LIN {X 0,Y 303.46,Z 323.911,A -85,B 0,C 180,E1 -16452.825,E2 -16452.825} C_VEL
LIN {X 0,Y 302.118,Z 332.035,A -85,B 0,C 180,E1 -16454.483,E2 -16454.483} C_VEL
LIN {X 0,Y 300.639,Z 339.994,A -85,B 0,C 180,E1 -16456.481,E2 -16456.481} C_VEL
LIN {X 0,Y 299.435,Z 346.378,A -85,B 0,C 180,E1 -16458.492,E2 -16458.492} C_VEL
LIN {X 0,Y 298.527,Z 351.434,A -85,B 0,C 180,E1 -16460.514,E2 -16460.514} C_VEL
LIN {X 0,Y 298.006,Z 354.562,A -85,B 0,C 180,E1 -16462.099,E2 -16462.099} C_VEL
LIN {X 0,Y 297.368,Z 358.253,A -85,B 0,C 180,E1 -16464.575,E2 -16464.575} C_VEL
LIN {X 0,Y 297.174,Z 359.637,A -85,B 0,C 180,E1 -16465.931,E2 -16465.931} C_VEL
LIN {X 0,Y 296.944,Z 361.227,A -85,B 0,C 180,E1 -16468.644,E2 -16468.644} C_VEL
LIN {X 0,Y 296.928,Z 361.456,A -85,B 0,C 180,E1 -16470,E2 -16470} C_VEL
LIN {X 0,Y 296.943,Z 361.266,A -85,B 0,C 180,E1 -16471.356,E2 -16471.356} C_VEL
LIN {X 0,Y 297.157,Z 359.726,A -85,B 0,C 180,E1 -16474.069,E2 -16474.069} C_VEL
LIN {X 0,Y 297.357,Z 358.38,A -85,B 0,C 180,E1 -16475.425,E2 -16475.425} C_VEL
LIN {X 0,Y 297.953,Z 354.9,A -85,B 0,C 180,E1 -16477.826,E2 -16477.826} C_VEL
LIN {X 0,Y 298.756,Z 350.121,A -85,B 0,C 180,E1 -16480.162,E2 -16480.162} C_VEL
LIN {X 0,Y 299.99,Z 343.715,A -85,B 0,C 180,E1 -16482.515,E2 -16482.515} C_VEL
LIN {X 0,Y 301.265,Z 336.671,A -85,B 0,C 180,E1 -16484.524,E2 -16484.524} C_VEL
LIN {X 0,Y 302.83,Z 327.889,A -85,B 0,C 180,E1 -16486.517,E2 -16486.517} C_VEL
LIN {X 0,Y 304.365,Z 318.867,A -85,B 0,C 180,E1 -16488.163,E2 -16488.163} C_VEL
LIN {X 0,Y 305.711,Z 308.49,A -85,B 0,C 180,E1 -16489.7,E2 -16489.7} C_VEL
LIN {X 0,Y 307.133,Z 297.75,A -85,B 0,C 180,E1 -16490.949,E2 -16490.949} C_VEL
LIN {X 0,Y 307.473,Z 294.559,A -85,B 0,C 180,E1 -16491.276,E2 -16491.276} C_VEL
LIN {X 0,Y 305.517,Z 284.175,A -85,B 0,C 180,E1 -16492.412,E2 -16492.412} C_VEL
LIN {X 0,Y 302.269,Z 271.951,A -85,B 0,C 180,E1 -16493.56,E2 -16493.56} C_VEL
LIN {X 0,Y 297.755,Z 258.35,A -85,B 0,C 180,E1 -16494.625,E2 -16494.625} C_VEL
LIN {X 0,Y 297.811,Z 255.408,A -85,B 0,C 180,E1 -16498.163,E2 -16498.163} C_VEL
LIN {X 0,Y 297.983,Z 252.472,A -85,B 0,C 180,E1 -16501.889,E2 -16501.889} C_VEL
LIN {X 0,Y 297.989,Z 251.752,A -85,B 0,C 180,E1 -16502.851,E2 -16502.851} C_VEL
LIN {X 0,Y 298.161,Z 251.347,A -85,B 0,C 180,E1 -16504.452,E2 -16504.452} C_VEL
LIN {X 0,Y 298.374,Z 251.321,A -85,B 0,C 180,E1 -16507.764,E2 -16507.764} C_VEL
LIN {X 0,Y 298.386,Z 251.316,A -85,B 0,C 180,E1 -16511.261,E2 -16511.261} C_VEL
LIN {X 0,Y 298.355,Z 251.319,A -85,B 0,C 180,E1 -16515.035,E2 -16515.035} C_VEL
LIN {X 0,Y 298.386,Z 251.315,A -85,B 0,C 180,E1 -16518.738,E2 -16518.738} C_VEL
LIN {X 0,Y 298.426,Z 251.311,A -85,B 0,C 180,E1 -16522.243,E2 -16522.243} C_VEL
LIN {X 0,Y 298.41,Z 251.315,A -85,B 0,C 180,E1 -16525.581,E2 -16525.581} C_VEL
LIN {X 0,Y 298.379,Z 251.314,A -85,B 0,C 180,E1 -16528.789,E2 -16528.789} C_VEL
LIN {X 0,Y 298.415,Z 251.312,A -85,B 0,C 180,E1 -16531.899,E2 -16531.899} C_VEL
LIN {X 0,Y 298.441,Z 251.308,A -85,B 0,C 180,E1 -16534.92,E2 -16534.92} C_VEL
LIN {X 0,Y 298.416,Z 251.31,A -85,B 0,C 180,E1 -16537.863,E2 -16537.863} C_VEL
LIN {X 0,Y 298.505,Z 251.301,A -85,B 0,C 180,E1 -16540.754,E2 -16540.754} C_VEL
LIN {X 0,Y 298.587,Z 251.292,A -85,B 0,C 180,E1 -16544.994,E2 -16544.994} C_VEL
LIN {X 0,Y 298.596,Z 251.291,A -85,B 0,C 180,E1 -16549.147,E2 -16549.147} C_VEL
LIN {X 0,Y 298.703,Z 251.276,A -85,B 0,C 180,E1 -16550.695,E2 -16550.695} C_VEL
LIN {X 0,Y 298.097,Z 251.352,A -85,B 0,C 180,E1 -16551.822,E2 -16551.822} C_VEL
LIN {X 0,Y 295.14,Z 251.719,A -85,B 0,C 180,E1 -16553.651,E2 -16553.651} C_VEL
LIN {X 0,Y 292.648,Z 252.03,A -85,B 0,C 180,E1 -16555.138,E2 -16555.138} C_VEL
LIN {X 0,Y 291.677,Z 252.151,A -85,B 0,C 180,E1 -16556.292,E2 -16556.292} C_VEL
LIN {X 0,Y 291.655,Z 252.151,A -85,B 0,C 180,E1 -16556.683,E2 -16556.683} C_VEL
LIN {X 0,Y 291.874,Z 252.13,A -85,B 0,C 180,E1 -16558.62,E2 -16558.62} C_VEL
LIN {X 0,Y 291.889,Z 252.124,A -85,B 0,C 180,E1 -16561.38,E2 -16561.38} C_VEL
LIN {X 0,Y 291.725,Z 252.145,A -85,B 0,C 180,E1 -16566.918,E2 -16566.918} C_VEL
LIN {X 0,Y 291.569,Z 252.164,A -85,B 0,C 180,E1 -16569.714,E2 -16569.714} C_VEL
LIN {X 0,Y 291.523,Z 252.172,A -85,B 0,C 180,E1 -16573.95,E2 -16573.95} C_VEL
LIN {X 0,Y 291.489,Z 252.174,A -85,B 0,C 180,E1 -16576.818,E2 -16576.818} C_VEL
LIN {X 0,Y 291.452,Z 252.182,A -85,B 0,C 180,E1 -16579.875,E2 -16579.875} C_VEL
LIN {X 0,Y 291.335,Z 252.197,A -85,B 0,C 180,E1 -16584.211,E2 -16584.211} C_VEL
LIN {X 0,Y 291.352,Z 252.196,A -85,B 0,C 180,E1 -16587.279,E2 -16587.279} C_VEL
LIN {X 0,Y 291.32,Z 252.199,A -85,B 0,C 180,E1 -16590.439,E2 -16590.439} C_VEL
LIN {X 0,Y 291.345,Z 252.197,A -85,B 0,C 180,E1 -16593.698,E2 -16593.698} C_VEL
LIN {X 0,Y 291.36,Z 252.193,A -85,B 0,C 180,E1 -16597.25,E2 -16597.25} C_VEL
LIN {X 0,Y 291.401,Z 252.404,A -85,B 0,C 180,E1 -16598.619,E2 -16598.619} C_VEL
LIN {X 0,Y 292.148,Z 256.598,A -85,B 0,C 180,E1 -16602.344,E2 -16602.344} C_VEL
LIN {X 0,Y 293.011,Z 261.073,A -85,B 0,C 180,E1 -16606.019,E2 -16606.019} C_VEL
LIN {X 0,Y 293.916,Z 266.185,A -85,B 0,C 180,E1 -16609.922,E2 -16609.922} C_VEL
LIN {X 0,Y 294.31,Z 269.06,A -85,B 0,C 180,E1 -16612.002,E2 -16612.002} C_VEL
LIN {X 0,Y 294.165,Z 272.478,A -85,B 0,C 180,E1 -16614.322,E2 -16614.322} C_VEL
LIN {X 0,Y 293.112,Z 278.393,A -85,B 0,C 180,E1 -16618.163,E2 -16618.163} C_VEL
LIN {X 0,Y 292.122,Z 284.445,A -85,B 0,C 180,E1 -16622.022,E2 -16622.022} C_VEL
LIN {X 0,Y 291.473,Z 288.992,A -85,B 0,C 180,E1 -16624.815,E2 -16624.815} C_VEL
LIN {X 0,Y 294.407,Z 302.447,A -85,B 0,C 180,E1 -16625.676,E2 -16625.676} C_VEL
LIN {X 0,Y 296.405,Z 315.779,A -85,B 0,C 180,E1 -16626.761,E2 -16626.761} C_VEL
LIN {X 0,Y 297.483,Z 327.947,A -85,B 0,C 180,E1 -16627.973,E2 -16627.973} C_VEL
LIN {X 0,Y 297.935,Z 338.759,A -85,B 0,C 180,E1 -16629.278,E2 -16629.278} C_VEL
LIN {X 0,Y 296.165,Z 349.684,A -85,B 0,C 180,E1 -16630.777,E2 -16630.777} C_VEL
LIN {X 0,Y 294.663,Z 358.572,A -85,B 0,C 180,E1 -16632.289,E2 -16632.289} C_VEL
LIN {X 0,Y 293.407,Z 366.829,A -85,B 0,C 180,E1 -16634.011,E2 -16634.011} C_VEL
LIN {X 0,Y 292.021,Z 374.897,A -85,B 0,C 180,E1 -16636.074,E2 -16636.074} C_VEL
LIN {X 0,Y 290.893,Z 381.371,A -85,B 0,C 180,E1 -16638.15,E2 -16638.15} C_VEL
LIN {X 0,Y 290.223,Z 386.529,A -85,B 0,C 180,E1 -16640.241,E2 -16640.241} C_VEL
LIN {X 0,Y 289.817,Z 390.543,A -85,B 0,C 180,E1 -16642.336,E2 -16642.336} C_VEL
LIN {X 0,Y 289.625,Z 393.516,A -85,B 0,C 180,E1 -16644.43,E2 -16644.43} C_VEL
LIN {X 0,Y 289.583,Z 394.933,A -85,B 0,C 180,E1 -16645.825,E2 -16645.825} C_VEL
LIN {X 0,Y 289.557,Z 395.944,A -85,B 0,C 180,E1 -16647.218,E2 -16647.218} C_VEL
LIN {X 0,Y 289.581,Z 396.564,A -85,B 0,C 180,E1 -16648.61,E2 -16648.61} C_VEL
LIN {X 0,Y 289.692,Z 396.788,A -85,B 0,C 180,E1 -16650,E2 -16650} C_VEL
LIN {X 0,Y 289.581,Z 396.559,A -85,B 0,C 180,E1 -16651.391,E2 -16651.391} C_VEL
LIN {X 0,Y 289.557,Z 395.938,A -85,B 0,C 180,E1 -16652.783,E2 -16652.783} C_VEL
LIN {X 0,Y 289.582,Z 394.924,A -85,B 0,C 180,E1 -16654.176,E2 -16654.176} C_VEL
LIN {X 0,Y 289.632,Z 393.206,A -85,B 0,C 180,E1 -16655.802,E2 -16655.802} C_VEL
LIN {X 0,Y 289.906,Z 389.275,A -85,B 0,C 180,E1 -16658.364,E2 -16658.364} C_VEL
LIN {X 0,Y 290.45,Z 384.885,A -85,B 0,C 180,E1 -16660.456,E2 -16660.456} C_VEL
LIN {X 0,Y 291.205,Z 379.299,A -85,B 0,C 180,E1 -16662.545,E2 -16662.545} C_VEL
LIN {X 0,Y 292.467,Z 372.352,A -85,B 0,C 180,E1 -16664.615,E2 -16664.615} C_VEL
LIN {X 0,Y 293.943,Z 363.661,A -85,B 0,C 180,E1 -16666.674,E2 -16666.674} C_VEL
LIN {X 0,Y 295.26,Z 354.749,A -85,B 0,C 180,E1 -16668.385,E2 -16668.385} C_VEL
LIN {X 0,Y 297.11,Z 343.814,A -85,B 0,C 180,E1 -16670.06,E2 -16670.06} C_VEL
LIN {X 0,Y 297.932,Z 338.625,A -85,B 0,C 180,E1 -16670.723,E2 -16670.723} C_VEL
LIN {X 0,Y 297.425,Z 327.766,A -85,B 0,C 180,E1 -16672.032,E2 -16672.032} C_VEL
LIN {X 0,Y 296.354,Z 315.227,A -85,B 0,C 180,E1 -16673.268,E2 -16673.268} C_VEL
LIN {X 0,Y 294.319,Z 301.984,A -85,B 0,C 180,E1 -16674.338,E2 -16674.338} C_VEL
LIN {X 0,Y 291.474,Z 288.763,A -85,B 0,C 180,E1 -16675.197,E2 -16675.197} C_VEL
LIN {X 0,Y 292.497,Z 282.092,A -85,B 0,C 180,E1 -16679.454,E2 -16679.454} C_VEL
LIN {X 0,Y 293.547,Z 275.913,A -85,B 0,C 180,E1 -16683.413,E2 -16683.413} C_VEL
LIN {X 0,Y 294.363,Z 270.985,A -85,B 0,C 180,E1 -16686.647,E2 -16686.647} C_VEL
LIN {X 0,Y 294.104,Z 267.282,A -85,B 0,C 180,E1 -16689.223,E2 -16689.223} C_VEL
LIN {X 0,Y 293.207,Z 262.122,A -85,B 0,C 180,E1 -16693.056,E2 -16693.056} C_VEL
LIN {X 0,Y 292.472,Z 258.342,A -85,B 0,C 180,E1 -16696.129,E2 -16696.129} C_VEL
LIN {X 0,Y 291.749,Z 254.528,A -85,B 0,C 180,E1 -16699.428,E2 -16699.428} C_VEL
LIN {X 0,Y 291.35,Z 252.192,A -85,B 0,C 180,E1 -16701.588,E2 -16701.588} C_VEL
LIN {X 0,Y 291.37,Z 252.191,A -85,B 0,C 180,E1 -16705.095,E2 -16705.095} C_VEL
LIN {X 0,Y 291.369,Z 252.19,A -85,B 0,C 180,E1 -16707.95,E2 -16707.95} C_VEL
LIN {X 0,Y 291.346,Z 252.192,A -85,B 0,C 180,E1 -16711.154,E2 -16711.154} C_VEL
LIN {X 0,Y 291.35,Z 252.196,A -85,B 0,C 180,E1 -16714.266,E2 -16714.266} C_VEL
LIN {X 0,Y 291.356,Z 252.192,A -85,B 0,C 180,E1 -16717.297,E2 -16717.297} C_VEL
LIN {X 0,Y 291.461,Z 252.182,A -85,B 0,C 180,E1 -16720.27,E2 -16720.27} C_VEL
LIN {X 0,Y 291.559,Z 252.166,A -85,B 0,C 180,E1 -16724.624,E2 -16724.624} C_VEL
LIN {X 0,Y 291.532,Z 252.169,A -85,B 0,C 180,E1 -16728.88,E2 -16728.88} C_VEL
LIN {X 0,Y 291.66,Z 252.157,A -85,B 0,C 180,E1 -16731.687,E2 -16731.687} C_VEL
LIN {X 0,Y 291.627,Z 252.157,A -85,B 0,C 180,E1 -16734.468,E2 -16734.468} C_VEL
LIN {X 0,Y 291.891,Z 252.124,A -85,B 0,C 180,E1 -16738.62,E2 -16738.62} C_VEL
LIN {X 0,Y 291.876,Z 252.129,A -85,B 0,C 180,E1 -16741.38,E2 -16741.38} C_VEL
LIN {X 0,Y 291.719,Z 252.146,A -85,B 0,C 180,E1 -16746.919,E2 -16746.919} C_VEL
LIN {X 0,Y 291.572,Z 252.165,A -85,B 0,C 180,E1 -16749.714,E2 -16749.714} C_VEL
LIN {X 0,Y 291.52,Z 252.17,A -85,B 0,C 180,E1 -16753.951,E2 -16753.951} C_VEL
LIN {X 0,Y 291.437,Z 252.184,A -85,B 0,C 180,E1 -16756.821,E2 -16756.821} C_VEL
LIN {X 0,Y 291.427,Z 252.181,A -85,B 0,C 180,E1 -16759.86,E2 -16759.86} C_VEL
LIN {X 0,Y 291.364,Z 252.19,A -85,B 0,C 180,E1 -16764.209,E2 -16764.209} C_VEL
LIN {X 0,Y 291.357,Z 252.191,A -85,B 0,C 180,E1 -16767.278,E2 -16767.278} C_VEL
LIN {X 0,Y 291.321,Z 252.199,A -85,B 0,C 180,E1 -16770.439,E2 -16770.439} C_VEL
LIN {X 0,Y 291.347,Z 252.192,A -85,B 0,C 180,E1 -16773.698,E2 -16773.698} C_VEL
LIN {X 0,Y 291.384,Z 252.187,A -85,B 0,C 180,E1 -16777.255,E2 -16777.255} C_VEL
LIN {X 0,Y 291.337,Z 252.195,A -85,B 0,C 180,E1 -16780.642,E2 -16780.642} C_VEL
LIN {X 0,Y 291.293,Z 252.2,A -85,B 0,C 180,E1 -16784.402,E2 -16784.402} C_VEL
LIN {X 0,Y 291.329,Z 252.196,A -85,B 0,C 180,E1 -16788.404,E2 -16788.404} C_VEL
LIN {X 0,Y 291.337,Z 252.193,A -85,B 0,C 180,E1 -16791.155,E2 -16791.155} C_VEL
LIN {X 0,Y 291.329,Z 252.193,A -85,B 0,C 180,E1 -16792.907,E2 -16792.907} C_VEL
LIN {X 0,Y 291.005,Z 252.237,A -85,B 0,C 180,E1 -16796.257,E2 -16796.257} C_VEL
LIN {X 0,Y 290.906,Z 254.487,A -85,B 0,C 180,E1 -16799.513,E2 -16799.513} C_VEL
LIN {X 0,Y 290.769,Z 257.655,A -85,B 0,C 180,E1 -16803.42,E2 -16803.42} C_VEL
LIN {X 0,Y 290.733,Z 258.839,A -85,B 0,C 180,E1 -16804.862,E2 -16804.862} C_VEL
LIN {X 0,Y 295.305,Z 272.378,A -85,B 0,C 180,E1 -16805.967,E2 -16805.967} C_VEL
LIN {X 0,Y 298.493,Z 284.073,A -85,B 0,C 180,E1 -16807.102,E2 -16807.102} C_VEL
LIN {X 0,Y 300.734,Z 295.59,A -85,B 0,C 180,E1 -16808.403,E2 -16808.403} C_VEL
LIN {X 0,Y 299.32,Z 306.86,A -85,B 0,C 180,E1 -16809.69,E2 -16809.69} C_VEL
LIN {X 0,Y 297.828,Z 317.602,A -85,B 0,C 180,E1 -16811.245,E2 -16811.245} C_VEL
LIN {X 0,Y 296.371,Z 326.109,A -85,B 0,C 180,E1 -16812.757,E2 -16812.757} C_VEL
LIN {X 0,Y 295.071,Z 333.933,A -85,B 0,C 180,E1 -16814.457,E2 -16814.457} C_VEL
LIN {X 0,Y 293.529,Z 341.587,A -85,B 0,C 180,E1 -16816.5,E2 -16816.5} C_VEL
LIN {X 0,Y 292.128,Z 348.604,A -85,B 0,C 180,E1 -16818.903,E2 -16818.903} C_VEL
LIN {X 0,Y 291.296,Z 353.268,A -85,B 0,C 180,E1 -16820.977,E2 -16820.977} C_VEL
LIN {X 0,Y 290.723,Z 356.832,A -85,B 0,C 180,E1 -16823.057,E2 -16823.057} C_VEL
LIN {X 0,Y 290.329,Z 358.68,A -85,B 0,C 180,E1 -16824.443,E2 -16824.443} C_VEL
LIN {X 0,Y 290.104,Z 360.064,A -85,B 0,C 180,E1 -16825.832,E2 -16825.832} C_VEL
LIN {X 0,Y 289.859,Z 361.654,A -85,B 0,C 180,E1 -16828.61,E2 -16828.61} C_VEL
LIN {X 0,Y 289.841,Z 361.882,A -85,B 0,C 180,E1 -16830,E2 -16830} C_VEL
LIN {X 0,Y 289.858,Z 361.692,A -85,B 0,C 180,E1 -16831.389,E2 -16831.389} C_VEL
LIN {X 0,Y 290.088,Z 360.152,A -85,B 0,C 180,E1 -16834.168,E2 -16834.168} C_VEL
LIN {X 0,Y 290.316,Z 358.805,A -85,B 0,C 180,E1 -16835.557,E2 -16835.557} C_VEL
LIN {X 0,Y 290.903,Z 355.549,A -85,B 0,C 180,E1 -16837.889,E2 -16837.889} C_VEL
LIN {X 0,Y 291.775,Z 350.547,A -85,B 0,C 180,E1 -16840.408,E2 -16840.408} C_VEL
LIN {X 0,Y 293.09,Z 344.139,A -85,B 0,C 180,E1 -16842.815,E2 -16842.815} C_VEL
LIN {X 0,Y 294.421,Z 337.095,A -85,B 0,C 180,E1 -16844.869,E2 -16844.869} C_VEL
LIN {X 0,Y 296.051,Z 328.312,A -85,B 0,C 180,E1 -16846.906,E2 -16846.906} C_VEL
LIN {X 0,Y 297.643,Z 319.29,A -85,B 0,C 180,E1 -16848.588,E2 -16848.588} C_VEL
LIN {X 0,Y 298.991,Z 309.413,A -85,B 0,C 180,E1 -16850.091,E2 -16850.091} C_VEL
LIN {X 0,Y 300.524,Z 298.171,A -85,B 0,C 180,E1 -16851.432,E2 -16851.432} C_VEL
LIN {X 0,Y 300.731,Z 294.989,A -85,B 0,C 180,E1 -16851.777,E2 -16851.777} C_VEL
LIN {X 0,Y 298.469,Z 283.823,A -85,B 0,C 180,E1 -16853.037,E2 -16853.037} C_VEL
LIN {X 0,Y 295.243,Z 272.161,A -85,B 0,C 180,E1 -16854.171,E2 -16854.171} C_VEL
LIN {X 0,Y 291.253,Z 260.862,A -85,B 0,C 180,E1 -16855.118,E2 -16855.118} C_VEL
LIN {X 0,Y 290.703,Z 258.773,A -85,B 0,C 180,E1 -16855.288,E2 -16855.288} C_VEL
LIN {X 0,Y 290.864,Z 255.325,A -85,B 0,C 180,E1 -16859.558,E2 -16859.558} C_VEL
LIN {X 0,Y 290.954,Z 253.239,A -85,B 0,C 180,E1 -16862.282,E2 -16862.282} C_VEL
LIN {X 0,Y 291.004,Z 252.239,A -85,B 0,C 180,E1 -16863.743,E2 -16863.743} C_VEL
LIN {X 0,Y 291.317,Z 252.199,A -85,B 0,C 180,E1 -16867.238,E2 -16867.238} C_VEL
LIN {X 0,Y 291.332,Z 252.196,A -85,B 0,C 180,E1 -16870.643,E2 -16870.643} C_VEL
LIN {X 0,Y 291.292,Z 252.201,A -85,B 0,C 180,E1 -16874.402,E2 -16874.402} C_VEL
LIN {X 0,Y 291.328,Z 252.195,A -85,B 0,C 180,E1 -16878.404,E2 -16878.404} C_VEL
LIN {X 0,Y 291.365,Z 252.19,A -85,B 0,C 180,E1 -16881.16,E2 -16881.16} C_VEL
LIN {X 0,Y 291.363,Z 252.19,A -85,B 0,C 180,E1 -16884.626,E2 -16884.626} C_VEL
LIN {X 0,Y 291.368,Z 252.19,A -85,B 0,C 180,E1 -16887.95,E2 -16887.95} C_VEL
LIN {X 0,Y 291.346,Z 252.194,A -85,B 0,C 180,E1 -16891.154,E2 -16891.154} C_VEL
LIN {X 0,Y 291.36,Z 252.189,A -85,B 0,C 180,E1 -16894.266,E2 -16894.266} C_VEL
LIN {X 0,Y 291.372,Z 252.191,A -85,B 0,C 180,E1 -16897.299,E2 -16897.299} C_VEL
LIN {X 0,Y 291.441,Z 252.18,A -85,B 0,C 180,E1 -16900.269,E2 -16900.269} C_VEL
LIN {X 0,Y 291.499,Z 252.174,A -85,B 0,C 180,E1 -16904.665,E2 -16904.665} C_VEL
LIN {X 0,Y 291.539,Z 252.17,A -85,B 0,C 180,E1 -16908.881,E2 -16908.881} C_VEL
LIN {X 0,Y 291.711,Z 252.146,A -85,B 0,C 180,E1 -16911.688,E2 -16911.688} C_VEL
LIN {X 0,Y 291.627,Z 252.159,A -85,B 0,C 180,E1 -16914.468,E2 -16914.468} C_VEL
LIN {X 0,Y 291.655,Z 252.151,A -85,B 0,C 180,E1 -16916.683,E2 -16916.683} C_VEL
LIN {X 0,Y 291.459,Z 252.178,A -85,B 0,C 180,E1 -16917.454,E2 -16917.454} C_VEL
LIN {X 0,Y 290.212,Z 252.337,A -85,B 0,C 180,E1 -16918.594,E2 -16918.594} C_VEL
LIN {X 0,Y 285.906,Z 252.87,A -85,B 0,C 180,E1 -16921.243,E2 -16921.243} C_VEL
LIN {X 0,Y 284.834,Z 253.006,A -85,B 0,C 180,E1 -16922.426,E2 -16922.426} C_VEL
LIN {X 0,Y 284.744,Z 253.015,A -85,B 0,C 180,E1 -16922.827,E2 -16922.827} C_VEL
LIN {X 0,Y 284.676,Z 253.023,A -85,B 0,C 180,E1 -16927.091,E2 -16927.091} C_VEL
LIN {X 0,Y 284.515,Z 253.044,A -85,B 0,C 180,E1 -16929.957,E2 -16929.957} C_VEL
LIN {X 0,Y 284.483,Z 253.049,A -85,B 0,C 180,E1 -16934.303,E2 -16934.303} C_VEL
LIN {X 0,Y 284.427,Z 253.054,A -85,B 0,C 180,E1 -16937.248,E2 -16937.248} C_VEL
LIN {X 0,Y 284.378,Z 253.063,A -85,B 0,C 180,E1 -16940.242,E2 -16940.242} C_VEL
LIN {X 0,Y 284.29,Z 253.074,A -85,B 0,C 180,E1 -16944.851,E2 -16944.851} C_VEL
LIN {X 0,Y 284.282,Z 253.078,A -85,B 0,C 180,E1 -16948.016,E2 -16948.016} C_VEL
LIN {X 0,Y 284.286,Z 253.078,A -85,B 0,C 180,E1 -16951.276,E2 -16951.276} C_VEL
LIN {X 0,Y 284.337,Z 253.069,A -85,B 0,C 180,E1 -16955.347,E2 -16955.347} C_VEL
LIN {X 0,Y 284.345,Z 253.209,A -85,B 0,C 180,E1 -16957.879,E2 -16957.879} C_VEL
LIN {X 0,Y 285.219,Z 258.045,A -85,B 0,C 180,E1 -16962.335,E2 -16962.335} C_VEL
LIN {X 0,Y 286.174,Z 263.074,A -85,B 0,C 180,E1 -16966.557,E2 -16966.557} C_VEL
LIN {X 0,Y 287.051,Z 268.111,A -85,B 0,C 180,E1 -16970.464,E2 -16970.464} C_VEL
LIN {X 0,Y 287.331,Z 271.836,A -85,B 0,C 180,E1 -16973.158,E2 -16973.158} C_VEL
LIN {X 0,Y 286.498,Z 276.801,A -85,B 0,C 180,E1 -16976.517,E2 -16976.517} C_VEL
LIN {X 0,Y 285.43,Z 282.827,A -85,B 0,C 180,E1 -16980.498,E2 -16980.498} C_VEL
LIN {X 0,Y 284.533,Z 288.393,A -85,B 0,C 180,E1 -16984.138,E2 -16984.138} C_VEL
LIN {X 0,Y 287.621,Z 302.816,A -85,B 0,C 180,E1 -16985.114,E2 -16985.114} C_VEL
LIN {X 0,Y 289.477,Z 314.636,A -85,B 0,C 180,E1 -16986.113,E2 -16986.113} C_VEL
LIN {X 0,Y 290.5,Z 325.712,A -85,B 0,C 180,E1 -16987.227,E2 -16987.227} C_VEL
LIN {X 0,Y 291.01,Z 336.89,A -85,B 0,C 180,E1 -16988.577,E2 -16988.577} C_VEL
LIN {X 0,Y 290.884,Z 340.948,A -85,B 0,C 180,E1 -16989.122,E2 -16989.122} C_VEL
LIN {X 0,Y 289.035,Z 351.408,A -85,B 0,C 180,E1 -16990.653,E2 -16990.653} C_VEL
LIN {X 0,Y 287.482,Z 360.33,A -85,B 0,C 180,E1 -16992.28,E2 -16992.28} C_VEL
LIN {X 0,Y 285.982,Z 369.281,A -85,B 0,C 180,E1 -16994.316,E2 -16994.316} C_VEL
LIN {X 0,Y 284.671,Z 376.764,A -85,B 0,C 180,E1 -16996.436,E2 -16996.436} C_VEL
LIN {X 0,Y 283.646,Z 382.781,A -85,B 0,C 180,E1 -16998.567,E2 -16998.567} C_VEL
LIN {X 0,Y 283.031,Z 387.55,A -85,B 0,C 180,E1 -17000.712,E2 -17000.712} C_VEL
LIN {X 0,Y 282.681,Z 391.202,A -85,B 0,C 180,E1 -17002.859,E2 -17002.859} C_VEL
LIN {X 0,Y 282.562,Z 393.089,A -85,B 0,C 180,E1 -17004.29,E2 -17004.29} C_VEL
LIN {X 0,Y 282.503,Z 394.506,A -85,B 0,C 180,E1 -17005.72,E2 -17005.72} C_VEL
LIN {X 0,Y 282.483,Z 395.518,A -85,B 0,C 180,E1 -17007.148,E2 -17007.148} C_VEL
LIN {X 0,Y 282.495,Z 396.137,A -85,B 0,C 180,E1 -17008.575,E2 -17008.575} C_VEL
LIN {X 0,Y 282.602,Z 396.361,A -85,B 0,C 180,E1 -17010,E2 -17010} C_VEL
LIN {X 0,Y 282.483,Z 395.511,A -85,B 0,C 180,E1 -17012.852,E2 -17012.852} C_VEL
LIN {X 0,Y 282.502,Z 394.496,A -85,B 0,C 180,E1 -17014.28,E2 -17014.28} C_VEL
LIN {X 0,Y 282.559,Z 392.986,A -85,B 0,C 180,E1 -17015.782,E2 -17015.782} C_VEL
LIN {X 0,Y 282.74,Z 390.089,A -85,B 0,C 180,E1 -17017.858,E2 -17017.858} C_VEL
LIN {X 0,Y 283.196,Z 386.065,A -85,B 0,C 180,E1 -17020.004,E2 -17020.004} C_VEL
LIN {X 0,Y 284.079,Z 379.888,A -85,B 0,C 180,E1 -17022.502,E2 -17022.502} C_VEL
LIN {X 0,Y 285.342,Z 373.165,A -85,B 0,C 180,E1 -17024.623,E2 -17024.623} C_VEL
LIN {X 0,Y 286.837,Z 364.828,A -85,B 0,C 180,E1 -17026.732,E2 -17026.732} C_VEL
LIN {X 0,Y 288.178,Z 356.278,A -85,B 0,C 180,E1 -17028.484,E2 -17028.484} C_VEL
LIN {X 0,Y 289.825,Z 346.923,A -85,B 0,C 180,E1 -17030.031,E2 -17030.031} C_VEL
LIN {X 0,Y 291.077,Z 339.515,A -85,B 0,C 180,E1 -17031.049,E2 -17031.049} C_VEL
LIN {X 0,Y 290.66,Z 328.144,A -85,B 0,C 180,E1 -17032.486,E2 -17032.486} C_VEL
LIN {X 0,Y 289.617,Z 315.766,A -85,B 0,C 180,E1 -17033.761,E2 -17033.761} C_VEL
LIN {X 0,Y 287.603,Z 302.612,A -85,B 0,C 180,E1 -17034.878,E2 -17034.878} C_VEL
LIN {X 0,Y 284.779,Z 290.047,A -85,B 0,C 180,E1 -17035.748,E2 -17035.748} C_VEL
LIN {X 0,Y 284.525,Z 288.292,A -85,B 0,C 180,E1 -17035.863,E2 -17035.863} C_VEL
LIN {X 0,Y 285.428,Z 282.785,A -85,B 0,C 180,E1 -17039.502,E2 -17039.502} C_VEL
LIN {X 0,Y 286.498,Z 276.76,A -85,B 0,C 180,E1 -17043.483,E2 -17043.483} C_VEL
LIN {X 0,Y 287.345,Z 271.792,A -85,B 0,C 180,E1 -17046.841,E2 -17046.841} C_VEL
LIN {X 0,Y 287.041,Z 268.049,A -85,B 0,C 180,E1 -17049.539,E2 -17049.539} C_VEL
LIN {X 0,Y 286.145,Z 263.016,A -85,B 0,C 180,E1 -17053.449,E2 -17053.449} C_VEL
LIN {X 0,Y 285.438,Z 259.423,A -85,B 0,C 180,E1 -17056.416,E2 -17056.416} C_VEL
LIN {X 0,Y 284.709,Z 255.313,A -85,B 0,C 180,E1 -17060.073,E2 -17060.073} C_VEL
LIN {X 0,Y 284.326,Z 253.071,A -85,B 0,C 180,E1 -17062.278,E2 -17062.278} C_VEL
LIN {X 0,Y 284.309,Z 253.07,A -85,B 0,C 180,E1 -17065.351,E2 -17065.351} C_VEL
LIN {X 0,Y 284.288,Z 253.075,A -85,B 0,C 180,E1 -17068.725,E2 -17068.725} C_VEL
LIN {X 0,Y 284.284,Z 253.074,A -85,B 0,C 180,E1 -17071.984,E2 -17071.984} C_VEL
LIN {X 0,Y 284.301,Z 253.074,A -85,B 0,C 180,E1 -17076.158,E2 -17076.158} C_VEL
LIN {X 0,Y 284.391,Z 253.062,A -85,B 0,C 180,E1 -17079.898,E2 -17079.898} C_VEL
LIN {X 0,Y 284.496,Z 253.047,A -85,B 0,C 180,E1 -17084.459,E2 -17084.459} C_VEL
LIN {X 0,Y 284.485,Z 253.047,A -85,B 0,C 180,E1 -17088.601,E2 -17088.601} C_VEL
LIN {X 0,Y 284.605,Z 253.034,A -85,B 0,C 180,E1 -17091.48,E2 -17091.48} C_VEL
LIN {X 0,Y 284.597,Z 253.033,A -85,B 0,C 180,E1 -17094.331,E2 -17094.331} C_VEL
LIN {X 0,Y 284.858,Z 253,A -85,B 0,C 180,E1 -17098.586,E2 -17098.586} C_VEL
LIN {X 0,Y 284.843,Z 253.005,A -85,B 0,C 180,E1 -17101.414,E2 -17101.414} C_VEL
LIN {X 0,Y 284.672,Z 253.025,A -85,B 0,C 180,E1 -17107.091,E2 -17107.091} C_VEL
LIN {X 0,Y 284.518,Z 253.042,A -85,B 0,C 180,E1 -17109.957,E2 -17109.957} C_VEL
LIN {X 0,Y 284.467,Z 253.049,A -85,B 0,C 180,E1 -17114.304,E2 -17114.304} C_VEL
LIN {X 0,Y 284.366,Z 253.063,A -85,B 0,C 180,E1 -17118.741,E2 -17118.741} C_VEL
LIN {X 0,Y 284.317,Z 253.067,A -85,B 0,C 180,E1 -17121.764,E2 -17121.764} C_VEL
LIN {X 0,Y 284.309,Z 253.071,A -85,B 0,C 180,E1 -17124.849,E2 -17124.849} C_VEL
LIN {X 0,Y 284.287,Z 253.072,A -85,B 0,C 180,E1 -17128.016,E2 -17128.016} C_VEL
LIN {X 0,Y 284.288,Z 253.071,A -85,B 0,C 180,E1 -17131.275,E2 -17131.275} C_VEL
LIN {X 0,Y 284.344,Z 253.063,A -85,B 0,C 180,E1 -17135.348,E2 -17135.348} C_VEL
LIN {X 0,Y 284.322,Z 253.071,A -85,B 0,C 180,E1 -17138.168,E2 -17138.168} C_VEL
LIN {X 0,Y 284.272,Z 253.075,A -85,B 0,C 180,E1 -17142.124,E2 -17142.124} C_VEL
LIN {X 0,Y 284.259,Z 253.078,A -85,B 0,C 180,E1 -17146.189,E2 -17146.189} C_VEL
LIN {X 0,Y 284.308,Z 253.072,A -85,B 0,C 180,E1 -17150.024,E2 -17150.024} C_VEL
LIN {X 0,Y 284.209,Z 253.083,A -85,B 0,C 180,E1 -17153.595,E2 -17153.595} C_VEL
LIN {X 0,Y 284.066,Z 253.1,A -85,B 0,C 180,E1 -17155.316,E2 -17155.316} C_VEL
LIN {X 0,Y 283.925,Z 253.915,A -85,B 0,C 180,E1 -17157.31,E2 -17157.31} C_VEL
LIN {X 0,Y 283.852,Z 256.161,A -85,B 0,C 180,E1 -17160.317,E2 -17160.317} C_VEL
LIN {X 0,Y 283.716,Z 259.303,A -85,B 0,C 180,E1 -17164.199,E2 -17164.199} C_VEL
LIN {X 0,Y 288.23,Z 272.476,A -85,B 0,C 180,E1 -17165.314,E2 -17165.314} C_VEL
LIN {X 0,Y 291.386,Z 283.527,A -85,B 0,C 180,E1 -17166.425,E2 -17166.425} C_VEL
LIN {X 0,Y 293.681,Z 294.335,A -85,B 0,C 180,E1 -17167.672,E2 -17167.672} C_VEL
LIN {X 0,Y 294.001,Z 297.599,A -85,B 0,C 180,E1 -17168.067,E2 -17168.067} C_VEL
LIN {X 0,Y 292.504,Z 308.573,A -85,B 0,C 180,E1 -17169.379,E2 -17169.379} C_VEL
LIN {X 0,Y 290.953,Z 319.086,A -85,B 0,C 180,E1 -17170.968,E2 -17170.968} C_VEL
LIN {X 0,Y 289.335,Z 328.221,A -85,B 0,C 180,E1 -17172.689,E2 -17172.689} C_VEL
LIN {X 0,Y 287.615,Z 337.091,A -85,B 0,C 180,E1 -17174.77,E2 -17174.77} C_VEL
LIN {X 0,Y 286.258,Z 344.22,A -85,B 0,C 180,E1 -17176.873,E2 -17176.873} C_VEL
LIN {X 0,Y 285.185,Z 349.032,A -85,B 0,C 180,E1 -17178.629,E2 -17178.629} C_VEL
LIN {X 0,Y 284.296,Z 353.696,A -85,B 0,C 180,E1 -17180.753,E2 -17180.753} C_VEL
LIN {X 0,Y 283.681,Z 357.261,A -85,B 0,C 180,E1 -17182.884,E2 -17182.884} C_VEL
LIN {X 0,Y 283.293,Z 359.106,A -85,B 0,C 180,E1 -17184.305,E2 -17184.305} C_VEL
LIN {X 0,Y 283.038,Z 360.491,A -85,B 0,C 180,E1 -17185.728,E2 -17185.728} C_VEL
LIN {X 0,Y 282.774,Z 362.081,A -85,B 0,C 180,E1 -17188.576,E2 -17188.576} C_VEL
LIN {X 0,Y 282.755,Z 362.309,A -85,B 0,C 180,E1 -17190,E2 -17190} C_VEL
LIN {X 0,Y 282.773,Z 362.119,A -85,B 0,C 180,E1 -17191.424,E2 -17191.424} C_VEL
LIN {X 0,Y 283.023,Z 360.578,A -85,B 0,C 180,E1 -17194.272,E2 -17194.272} C_VEL
LIN {X 0,Y 283.277,Z 359.231,A -85,B 0,C 180,E1 -17195.695,E2 -17195.695} C_VEL
LIN {X 0,Y 283.861,Z 356.17,A -85,B 0,C 180,E1 -17197.967,E2 -17197.967} C_VEL
LIN {X 0,Y 284.516,Z 352.521,A -85,B 0,C 180,E1 -17199.957,E2 -17199.957} C_VEL
LIN {X 0,Y 285.511,Z 347.533,A -85,B 0,C 180,E1 -17202.077,E2 -17202.077} C_VEL
LIN {X 0,Y 286.802,Z 341.244,A -85,B 0,C 180,E1 -17204.184,E2 -17204.184} C_VEL
LIN {X 0,Y 288.356,Z 333.369,A -85,B 0,C 180,E1 -17206.277,E2 -17206.277} C_VEL
LIN {X 0,Y 290.263,Z 323.562,A -85,B 0,C 180,E1 -17208.346,E2 -17208.346} C_VEL
LIN {X 0,Y 291.74,Z 314.202,A -85,B 0,C 180,E1 -17209.93,E2 -17209.93} C_VEL
LIN {X 0,Y 293.156,Z 304.481,A -85,B 0,C 180,E1 -17211.26,E2 -17211.26} C_VEL
LIN {X 0,Y 294.08,Z 297.023,A -85,B 0,C 180,E1 -17212.111,E2 -17212.111} C_VEL
LIN {X 0,Y 292.019,Z 285.961,A -85,B 0,C 180,E1 -17213.429,E2 -17213.429} C_VEL
LIN {X 0,Y 288.746,Z 274.048,A -85,B 0,C 180,E1 -17214.657,E2 -17214.657} C_VEL
LIN {X 0,Y 284.567,Z 262.01,A -85,B 0,C 180,E1 -17215.72,E2 -17215.72} C_VEL
LIN {X 0,Y 283.698,Z 259.206,A -85,B 0,C 180,E1 -17215.97,E2 -17215.97} C_VEL
LIN {X 0,Y 283.868,Z 256.064,A -85,B 0,C 180,E1 -17219.942,E2 -17219.942} C_VEL
LIN {X 0,Y 283.932,Z 253.791,A -85,B 0,C 180,E1 -17222.994,E2 -17222.994} C_VEL
LIN {X 0,Y 284.126,Z 253.093,A -85,B 0,C 180,E1 -17225.286,E2 -17225.286} C_VEL
LIN {X 0,Y 284.268,Z 253.079,A -85,B 0,C 180,E1 -17228.176,E2 -17228.176} C_VEL
LIN {X 0,Y 284.273,Z 253.075,A -85,B 0,C 180,E1 -17231.875,E2 -17231.875} C_VEL
LIN {X 0,Y 284.257,Z 253.075,A -85,B 0,C 180,E1 -17236.189,E2 -17236.189} C_VEL
LIN {X 0,Y 284.308,Z 253.072,A -85,B 0,C 180,E1 -17240.024,E2 -17240.024} C_VEL
LIN {X 0,Y 284.336,Z 253.068,A -85,B 0,C 180,E1 -17243.614,E2 -17243.614} C_VEL
LIN {X 0,Y 284.308,Z 253.07,A -85,B 0,C 180,E1 -17247.19,E2 -17247.19} C_VEL
LIN {X 0,Y 284.339,Z 253.065,A -85,B 0,C 180,E1 -17250.374,E2 -17250.374} C_VEL
LIN {X 0,Y 284.307,Z 253.071,A -85,B 0,C 180,E1 -17253.579,E2 -17253.579} C_VEL
LIN {X 0,Y 284.33,Z 253.067,A -85,B 0,C 180,E1 -17256.704,E2 -17256.704} C_VEL
LIN {X 0,Y 284.378,Z 253.06,A -85,B 0,C 180,E1 -17259.904,E2 -17259.904} C_VEL
LIN {X 0,Y 284.448,Z 253.052,A -85,B 0,C 180,E1 -17264.492,E2 -17264.492} C_VEL
LIN {X 0,Y 284.491,Z 253.048,A -85,B 0,C 180,E1 -17268.601,E2 -17268.601} C_VEL
LIN {X 0,Y 284.661,Z 253.025,A -85,B 0,C 180,E1 -17271.481,E2 -17271.481} C_VEL
LIN {X 0,Y 284.599,Z 253.033,A -85,B 0,C 180,E1 -17274.331,E2 -17274.331} C_VEL
LIN {X 0,Y 284.841,Z 253.006,A -85,B 0,C 180,E1 -17278.586,E2 -17278.586} C_VEL
LIN {X 0,Y 284.856,Z 253.001,A -85,B 0,C 180,E1 -17281.414,E2 -17281.414} C_VEL
LIN {X 0,Y 284.744,Z 253.015,A -85,B 0,C 180,E1 -17282.827,E2 -17282.827} C_VEL
LIN {X 0,Y 284.082,Z 253.104,A -85,B 0,C 180,E1 -17284.006,E2 -17284.006} C_VEL
LIN {X 0,Y 281.259,Z 253.458,A -85,B 0,C 180,E1 -17285.928,E2 -17285.928} C_VEL
LIN {X 0,Y 277.955,Z 253.864,A -85,B 0,C 180,E1 -17288.288,E2 -17288.288} C_VEL
LIN {X 0,Y 277.557,Z 253.908,A -85,B 0,C 180,E1 -17289.105,E2 -17289.105} C_VEL
LIN {X 0,Y 277.417,Z 253.926,A -85,B 0,C 180,E1 -17293.18,E2 -17293.18} C_VEL
LIN {X 0,Y 277.408,Z 253.932,A -85,B 0,C 180,E1 -17296.181,E2 -17296.181} C_VEL
LIN {X 0,Y 277.321,Z 253.942,A -85,B 0,C 180,E1 -17300.335,E2 -17300.335} C_VEL
LIN {X 0,Y 277.242,Z 253.954,A -85,B 0,C 180,E1 -17304.134,E2 -17304.134} C_VEL
LIN {X 0,Y 277.268,Z 253.951,A -85,B 0,C 180,E1 -17307.482,E2 -17307.482} C_VEL
LIN {X 0,Y 277.248,Z 253.952,A -85,B 0,C 180,E1 -17310.473,E2 -17310.473} C_VEL
LIN {X 0,Y 277.247,Z 253.954,A -85,B 0,C 180,E1 -17313.896,E2 -17313.896} C_VEL
LIN {X 0,Y 277.284,Z 254.117,A -85,B 0,C 180,E1 -17317.24,E2 -17317.24} C_VEL
LIN {X 0,Y 277.989,Z 258.141,A -85,B 0,C 180,E1 -17321.096,E2 -17321.096} C_VEL
LIN {X 0,Y 278.878,Z 262.672,A -85,B 0,C 180,E1 -17325.12,E2 -17325.12} C_VEL
LIN {X 0,Y 279.783,Z 267.707,A -85,B 0,C 180,E1 -17329.224,E2 -17329.224} C_VEL
LIN {X 0,Y 280.27,Z 271.468,A -85,B 0,C 180,E1 -17332.095,E2 -17332.095} C_VEL
LIN {X 0,Y 280.272,Z 273.209,A -85,B 0,C 180,E1 -17333.362,E2 -17333.362} C_VEL
LIN {X 0,Y 279.47,Z 277.587,A -85,B 0,C 180,E1 -17336.41,E2 -17336.41} C_VEL
LIN {X 0,Y 278.365,Z 283.595,A -85,B 0,C 180,E1 -17340.506,E2 -17340.506} C_VEL
LIN {X 0,Y 277.615,Z 287.971,A -85,B 0,C 180,E1 -17343.454,E2 -17343.454} C_VEL
LIN {X 0,Y 280.584,Z 301.42,A -85,B 0,C 180,E1 -17344.385,E2 -17344.385} C_VEL
LIN {X 0,Y 282.617,Z 313.885,A -85,B 0,C 180,E1 -17345.469,E2 -17345.469} C_VEL
LIN {X 0,Y 283.793,Z 326.564,A -85,B 0,C 180,E1 -17346.796,E2 -17346.796} C_VEL
LIN {X 0,Y 284.215,Z 337.882,A -85,B 0,C 180,E1 -17348.228,E2 -17348.228} C_VEL
LIN {X 0,Y 284.025,Z 341.821,A -85,B 0,C 180,E1 -17348.784,E2 -17348.784} C_VEL
LIN {X 0,Y 282.119,Z 352.026,A -85,B 0,C 180,E1 -17350.348,E2 -17350.348} C_VEL
LIN {X 0,Y 280.403,Z 361.397,A -85,B 0,C 180,E1 -17352.158,E2 -17352.158} C_VEL
LIN {X 0,Y 279.132,Z 368.854,A -85,B 0,C 180,E1 -17353.921,E2 -17353.921} C_VEL
LIN {X 0,Y 277.716,Z 376.335,A -85,B 0,C 180,E1 -17356.089,E2 -17356.089} C_VEL
LIN {X 0,Y 276.63,Z 382.351,A -85,B 0,C 180,E1 -17358.273,E2 -17358.273} C_VEL
LIN {X 0,Y 275.985,Z 387.121,A -85,B 0,C 180,E1 -17360.473,E2 -17360.473} C_VEL
LIN {X 0,Y 275.61,Z 390.773,A -85,B 0,C 180,E1 -17362.675,E2 -17362.675} C_VEL
LIN {X 0,Y 275.49,Z 392.751,A -85,B 0,C 180,E1 -17364.227,E2 -17364.227} C_VEL
LIN {X 0,Y 275.412,Z 395.092,A -85,B 0,C 180,E1 -17367.075,E2 -17367.075} C_VEL
LIN {X 0,Y 275.413,Z 395.71,A -85,B 0,C 180,E1 -17368.538,E2 -17368.538} C_VEL
LIN {X 0,Y 275.513,Z 395.934,A -85,B 0,C 180,E1 -17370,E2 -17370} C_VEL
LIN {X 0,Y 275.412,Z 395.084,A -85,B 0,C 180,E1 -17372.926,E2 -17372.926} C_VEL
LIN {X 0,Y 275.446,Z 392.827,A -85,B 0,C 180,E1 -17375.682,E2 -17375.682} C_VEL
LIN {X 0,Y 275.698,Z 389.66,A -85,B 0,C 180,E1 -17378.06,E2 -17378.06} C_VEL
LIN {X 0,Y 276.182,Z 385.634,A -85,B 0,C 180,E1 -17380.261,E2 -17380.261} C_VEL
LIN {X 0,Y 277.096,Z 379.456,A -85,B 0,C 180,E1 -17382.823,E2 -17382.823} C_VEL
LIN {X 0,Y 278.435,Z 372.733,A -85,B 0,C 180,E1 -17384.995,E2 -17384.995} C_VEL
LIN {X 0,Y 279.999,Z 364.395,A -85,B 0,C 180,E1 -17387.153,E2 -17387.153} C_VEL
LIN {X 0,Y 281.401,Z 355.844,A -85,B 0,C 180,E1 -17388.946,E2 -17388.946} C_VEL
LIN {X 0,Y 283.335,Z 345.31,A -85,B 0,C 180,E1 -17390.7,E2 -17390.7} C_VEL
LIN {X 0,Y 284.216,Z 340.379,A -85,B 0,C 180,E1 -17391.392,E2 -17391.392} C_VEL
LIN {X 0,Y 283.92,Z 329.55,A -85,B 0,C 180,E1 -17392.832,E2 -17392.832} C_VEL
LIN {X 0,Y 283.094,Z 317.876,A -85,B 0,C 180,E1 -17394.121,E2 -17394.121} C_VEL
LIN {X 0,Y 281.224,Z 304.788,A -85,B 0,C 180,E1 -17395.314,E2 -17395.314} C_VEL
LIN {X 0,Y 278.295,Z 290.982,A -85,B 0,C 180,E1 -17396.335,E2 -17396.335} C_VEL
LIN {X 0,Y 277.61,Z 287.931,A -85,B 0,C 180,E1 -17396.526,E2 -17396.526} C_VEL
LIN {X 0,Y 278.726,Z 281.371,A -85,B 0,C 180,E1 -17400.985,E2 -17400.985} C_VEL
LIN {X 0,Y 279.966,Z 275.119,A -85,B 0,C 180,E1 -17405.266,E2 -17405.266} C_VEL
LIN {X 0,Y 280.314,Z 272.656,A -85,B 0,C 180,E1 -17406.994,E2 -17406.994} C_VEL
LIN {X 0,Y 280,Z 268.922,A -85,B 0,C 180,E1 -17409.795,E2 -17409.795} C_VEL
LIN {X 0,Y 279.01,Z 263.545,A -85,B 0,C 180,E1 -17414.087,E2 -17414.087} C_VEL
LIN {X 0,Y 278.206,Z 259.067,A -85,B 0,C 180,E1 -17417.997,E2 -17417.997} C_VEL
LIN {X 0,Y 277.324,Z 254.306,A -85,B 0,C 180,E1 -17422.54,E2 -17422.54} C_VEL
LIN {X 0,Y 277.261,Z 253.95,A -85,B 0,C 180,E1 -17422.982,E2 -17422.982} C_VEL
LIN {X 0,Y 277.255,Z 253.952,A -85,B 0,C 180,E1 -17426.773,E2 -17426.773} C_VEL
LIN {X 0,Y 277.264,Z 253.948,A -85,B 0,C 180,E1 -17429.539,E2 -17429.539} C_VEL
LIN {X 0,Y 277.292,Z 253.945,A -85,B 0,C 180,E1 -17432.857,E2 -17432.857} C_VEL
LIN {X 0,Y 277.263,Z 253.951,A -85,B 0,C 180,E1 -17436.073,E2 -17436.073} C_VEL
LIN {X 0,Y 277.346,Z 253.938,A -85,B 0,C 180,E1 -17440.766,E2 -17440.766} C_VEL
LIN {X 0,Y 277.438,Z 253.926,A -85,B 0,C 180,E1 -17445.326,E2 -17445.326} C_VEL
LIN {X 0,Y 277.46,Z 253.925,A -85,B 0,C 180,E1 -17449.787,E2 -17449.787} C_VEL
LIN {X 0,Y 277.627,Z 253.9,A -85,B 0,C 180,E1 -17452.728,E2 -17452.728} C_VEL
LIN {X 0,Y 277.824,Z 253.876,A -85,B 0,C 180,E1 -17458.551,E2 -17458.551} C_VEL
LIN {X 0,Y 277.81,Z 253.882,A -85,B 0,C 180,E1 -17461.45,E2 -17461.45} C_VEL
LIN {X 0,Y 277.627,Z 253.905,A -85,B 0,C 180,E1 -17467.272,E2 -17467.272} C_VEL
LIN {X 0,Y 277.461,Z 253.921,A -85,B 0,C 180,E1 -17470.213,E2 -17470.213} C_VEL
LIN {X 0,Y 277.413,Z 253.929,A -85,B 0,C 180,E1 -17474.675,E2 -17474.675} C_VEL
LIN {X 0,Y 277.321,Z 253.941,A -85,B 0,C 180,E1 -17479.236,E2 -17479.236} C_VEL
LIN {X 0,Y 277.286,Z 253.943,A -85,B 0,C 180,E1 -17483.925,E2 -17483.925} C_VEL
LIN {X 0,Y 277.273,Z 253.945,A -85,B 0,C 180,E1 -17487.483,E2 -17487.483} C_VEL
LIN {X 0,Y 277.251,Z 253.951,A -85,B 0,C 180,E1 -17490.473,E2 -17490.473} C_VEL
LIN {X 0,Y 277.25,Z 253.949,A -85,B 0,C 180,E1 -17493.896,E2 -17493.896} C_VEL
LIN {X 0,Y 277.275,Z 253.945,A -85,B 0,C 180,E1 -17497.468,E2 -17497.468} C_VEL
LIN {X 0,Y 277.213,Z 253.953,A -85,B 0,C 180,E1 -17501.236,E2 -17501.236} C_VEL
LIN {X 0,Y 277.204,Z 253.953,A -85,B 0,C 180,E1 -17505.226,E2 -17505.226} C_VEL
LIN {X 0,Y 277.225,Z 253.953,A -85,B 0,C 180,E1 -17509.512,E2 -17509.512} C_VEL
LIN {X 0,Y 277.201,Z 253.954,A -85,B 0,C 180,E1 -17512.52,E2 -17512.52} C_VEL
LIN {X 0,Y 276.94,Z 254.114,A -85,B 0,C 180,E1 -17516.061,E2 -17516.061} C_VEL
LIN {X 0,Y 276.845,Z 256.737,A -85,B 0,C 180,E1 -17519.67,E2 -17519.67} C_VEL
LIN {X 0,Y 276.711,Z 259.714,A -85,B 0,C 180,E1 -17523.488,E2 -17523.488} C_VEL
LIN {X 0,Y 278.681,Z 265.314,A -85,B 0,C 180,E1 -17523.95,E2 -17523.95} C_VEL
LIN {X 0,Y 282.255,Z 275.958,A -85,B 0,C 180,E1 -17524.957,E2 -17524.957} C_VEL
LIN {X 0,Y 285.27,Z 287.137,A -85,B 0,C 180,E1 -17526.174,E2 -17526.174} C_VEL
LIN {X 0,Y 287.383,Z 298.035,A -85,B 0,C 180,E1 -17527.535,E2 -17527.535} C_VEL
LIN {X 0,Y 285.856,Z 309.198,A -85,B 0,C 180,E1 -17528.905,E2 -17528.905} C_VEL
LIN {X 0,Y 284.273,Z 319.516,A -85,B 0,C 180,E1 -17530.503,E2 -17530.503} C_VEL
LIN {X 0,Y 282.59,Z 328.65,A -85,B 0,C 180,E1 -17532.262,E2 -17532.262} C_VEL
LIN {X 0,Y 280.792,Z 337.519,A -85,B 0,C 180,E1 -17534.391,E2 -17534.391} C_VEL
LIN {X 0,Y 279.376,Z 344.648,A -85,B 0,C 180,E1 -17536.544,E2 -17536.544} C_VEL
LIN {X 0,Y 278.253,Z 349.46,A -85,B 0,C 180,E1 -17538.342,E2 -17538.342} C_VEL
LIN {X 0,Y 277.299,Z 354.125,A -85,B 0,C 180,E1 -17540.518,E2 -17540.518} C_VEL
LIN {X 0,Y 276.646,Z 357.689,A -85,B 0,C 180,E1 -17542.702,E2 -17542.702} C_VEL
LIN {X 0,Y 276.259,Z 359.533,A -85,B 0,C 180,E1 -17544.159,E2 -17544.159} C_VEL
LIN {X 0,Y 275.976,Z 360.919,A -85,B 0,C 180,E1 -17545.618,E2 -17545.618} C_VEL
LIN {X 0,Y 275.689,Z 362.508,A -85,B 0,C 180,E1 -17548.539,E2 -17548.539} C_VEL
LIN {X 0,Y 275.668,Z 362.736,A -85,B 0,C 180,E1 -17550,E2 -17550} C_VEL
LIN {X 0,Y 275.688,Z 362.546,A -85,B 0,C 180,E1 -17551.461,E2 -17551.461} C_VEL
LIN {X 0,Y 275.961,Z 361.004,A -85,B 0,C 180,E1 -17554.382,E2 -17554.382} C_VEL
LIN {X 0,Y 276.241,Z 359.656,A -85,B 0,C 180,E1 -17555.841,E2 -17555.841} C_VEL
LIN {X 0,Y 276.805,Z 356.809,A -85,B 0,C 180,E1 -17558.026,E2 -17558.026} C_VEL
LIN {X 0,Y 277.537,Z 352.947,A -85,B 0,C 180,E1 -17560.21,E2 -17560.21} C_VEL
LIN {X 0,Y 278.595,Z 347.957,A -85,B 0,C 180,E1 -17562.382,E2 -17562.382} C_VEL
LIN {X 0,Y 279.927,Z 341.669,A -85,B 0,C 180,E1 -17564.54,E2 -17564.54} C_VEL
LIN {X 0,Y 281.544,Z 333.794,A -85,B 0,C 180,E1 -17566.682,E2 -17566.682} C_VEL
LIN {X 0,Y 283.556,Z 323.985,A -85,B 0,C 180,E1 -17568.796,E2 -17568.796} C_VEL
LIN {X 0,Y 285.256,Z 313.577,A -85,B 0,C 180,E1 -17570.572,E2 -17570.572} C_VEL
LIN {X 0,Y 286.81,Z 303.482,A -85,B 0,C 180,E1 -17571.943,E2 -17571.943} C_VEL
LIN {X 0,Y 287.362,Z 297.455,A -85,B 0,C 180,E1 -17572.656,E2 -17572.656} C_VEL
LIN {X 0,Y 284.937,Z 285.485,A -85,B 0,C 180,E1 -17574.131,E2 -17574.131} C_VEL
LIN {X 0,Y 281.434,Z 273.176,A -85,B 0,C 180,E1 -17575.431,E2 -17575.431} C_VEL
LIN {X 0,Y 276.822,Z 260.336,A -85,B 0,C 180,E1 -17576.592,E2 -17576.592} C_VEL
LIN {X 0,Y 276.701,Z 259.686,A -85,B 0,C 180,E1 -17576.632,E2 -17576.632} C_VEL
LIN {X 0,Y 276.845,Z 256.696,A -85,B 0,C 180,E1 -17580.512,E2 -17580.512} C_VEL
LIN {X 0,Y 276.939,Z 254.209,A -85,B 0,C 180,E1 -17583.938,E2 -17583.938} C_VEL
LIN {X 0,Y 277.111,Z 253.969,A -85,B 0,C 180,E1 -17585.75,E2 -17585.75} C_VEL
LIN {X 0,Y 277.222,Z 253.954,A -85,B 0,C 180,E1 -17589.33,E2 -17589.33} C_VEL
LIN {X 0,Y 277.211,Z 253.953,A -85,B 0,C 180,E1 -17593.198,E2 -17593.198} C_VEL
LIN {X 0,Y 277.216,Z 253.95,A -85,B 0,C 180,E1 -17597.325,E2 -17597.325} C_VEL
LIN {X 0,Y 277.272,Z 253.948,A -85,B 0,C 180,E1 -17601.791,E2 -17601.791} C_VEL
LIN {X 0,Y 277.287,Z 253.944,A -85,B 0,C 180,E1 -17604.342,E2 -17604.342} C_VEL
LIN {X 0,Y 277.242,Z 253.95,A -85,B 0,C 180,E1 -17607.836,E2 -17607.836} C_VEL
LIN {X 0,Y 277.241,Z 253.951,A -85,B 0,C 180,E1 -17611.207,E2 -17611.207} C_VEL
LIN {X 0,Y 277.248,Z 253.947,A -85,B 0,C 180,E1 -17614.473,E2 -17614.473} C_VEL
LIN {X 0,Y 277.265,Z 253.945,A -85,B 0,C 180,E1 -17617.653,E2 -17617.653} C_VEL
LIN {X 0,Y 277.319,Z 253.941,A -85,B 0,C 180,E1 -17620.764,E2 -17620.764} C_VEL
LIN {X 0,Y 277.411,Z 253.928,A -85,B 0,C 180,E1 -17625.324,E2 -17625.324} C_VEL
LIN {X 0,Y 277.509,Z 253.915,A -85,B 0,C 180,E1 -17629.789,E2 -17629.789} C_VEL
LIN {X 0,Y 277.655,Z 253.899,A -85,B 0,C 180,E1 -17632.729,E2 -17632.729} C_VEL
LIN {X 0,Y 277.808,Z 253.882,A -85,B 0,C 180,E1 -17638.55,E2 -17638.55} C_VEL
LIN {X 0,Y 277.822,Z 253.877,A -85,B 0,C 180,E1 -17641.449,E2 -17641.449} C_VEL
LIN {X 0,Y 277.63,Z 253.9,A -85,B 0,C 180,E1 -17647.271,E2 -17647.271} C_VEL
LIN {X 0,Y 277.557,Z 253.908,A -85,B 0,C 180,E1 -17649.105,E2 -17649.105} C_VEL
LIN {X 0,Y 276.781,Z 254.009,A -85,B 0,C 180,E1 -17650.314,E2 -17650.314} C_VEL
LIN {X 0,Y 273.889,Z 254.368,A -85,B 0,C 180,E1 -17652.285,E2 -17652.285} C_VEL
LIN {X 0,Y 271.497,Z 254.666,A -85,B 0,C 180,E1 -17653.886,E2 -17653.886} C_VEL
LIN {X 0,Y 270.472,Z 254.791,A -85,B 0,C 180,E1 -17655.127,E2 -17655.127} C_VEL
LIN {X 0,Y 270.385,Z 254.802,A -85,B 0,C 180,E1 -17655.547,E2 -17655.547} C_VEL
LIN {X 0,Y 270.291,Z 254.817,A -85,B 0,C 180,E1 -17659.756,E2 -17659.756} C_VEL
LIN {X 0,Y 270.18,Z 254.832,A -85,B 0,C 180,E1 -17664.595,E2 -17664.595} C_VEL
LIN {X 0,Y 270.198,Z 254.834,A -85,B 0,C 180,E1 -17667.917,E2 -17667.917} C_VEL
LIN {X 0,Y 270.174,Z 254.837,A -85,B 0,C 180,E1 -17671.35,E2 -17671.35} C_VEL
LIN {X 0,Y 270.199,Z 254.83,A -85,B 0,C 180,E1 -17674.906,E2 -17674.906} C_VEL
LIN {X 0,Y 270.258,Z 254.981,A -85,B 0,C 180,E1 -17676.51,E2 -17676.51} C_VEL
LIN {X 0,Y 270.905,Z 258.911,A -85,B 0,C 180,E1 -17680.434,E2 -17680.434} C_VEL
LIN {X 0,Y 271.728,Z 263.092,A -85,B 0,C 180,E1 -17684.293,E2 -17684.293} C_VEL
LIN {X 0,Y 272.596,Z 267.903,A -85,B 0,C 180,E1 -17688.389,E2 -17688.389} C_VEL
LIN {X 0,Y 273.077,Z 270.574,A -85,B 0,C 180,E1 -17690.542,E2 -17690.542} C_VEL
LIN {X 0,Y 273.273,Z 273.6,A -85,B 0,C 180,E1 -17692.869,E2 -17692.869} C_VEL
LIN {X 0,Y 272.665,Z 277.334,A -85,B 0,C 180,E1 -17695.569,E2 -17695.569} C_VEL
LIN {X 0,Y 271.483,Z 283.172,A -85,B 0,C 180,E1 -17699.682,E2 -17699.682} C_VEL
LIN {X 0,Y 270.691,Z 287.527,A -85,B 0,C 180,E1 -17702.72,E2 -17702.72} C_VEL
LIN {X 0,Y 273.761,Z 301.252,A -85,B 0,C 180,E1 -17703.717,E2 -17703.717} C_VEL
LIN {X 0,Y 275.802,Z 313.44,A -85,B 0,C 180,E1 -17704.821,E2 -17704.821} C_VEL
LIN {X 0,Y 277.002,Z 326.091,A -85,B 0,C 180,E1 -17706.189,E2 -17706.189} C_VEL
LIN {X 0,Y 277.417,Z 337.444,A -85,B 0,C 180,E1 -17707.666,E2 -17707.666} C_VEL
LIN {X 0,Y 277.172,Z 342.657,A -85,B 0,C 180,E1 -17708.428,E2 -17708.428} C_VEL
LIN {X 0,Y 275.009,Z 353.563,A -85,B 0,C 180,E1 -17710.208,E2 -17710.208} C_VEL
LIN {X 0,Y 273.303,Z 362.651,A -85,B 0,C 180,E1 -17712.075,E2 -17712.075} C_VEL
LIN {X 0,Y 271.987,Z 369.793,A -85,B 0,C 180,E1 -17713.873,E2 -17713.873} C_VEL
LIN {X 0,Y 270.593,Z 377.032,A -85,B 0,C 180,E1 -17716.099,E2 -17716.099} C_VEL
LIN {X 0,Y 269.63,Z 381.922,A -85,B 0,C 180,E1 -17717.964,E2 -17717.964} C_VEL
LIN {X 0,Y 268.961,Z 386.693,A -85,B 0,C 180,E1 -17720.221,E2 -17720.221} C_VEL
LIN {X 0,Y 268.539,Z 390.345,A -85,B 0,C 180,E1 -17722.481,E2 -17722.481} C_VEL
LIN {X 0,Y 268.415,Z 392.497,A -85,B 0,C 180,E1 -17724.25,E2 -17724.25} C_VEL
LIN {X 0,Y 268.341,Z 394.666,A -85,B 0,C 180,E1 -17726.998,E2 -17726.998} C_VEL
LIN {X 0,Y 268.333,Z 395.284,A -85,B 0,C 180,E1 -17728.499,E2 -17728.499} C_VEL
LIN {X 0,Y 268.425,Z 395.507,A -85,B 0,C 180,E1 -17730,E2 -17730} C_VEL
LIN {X 0,Y 268.341,Z 394.657,A -85,B 0,C 180,E1 -17733.003,E2 -17733.003} C_VEL
LIN {X 0,Y 268.357,Z 392.602,A -85,B 0,C 180,E1 -17735.626,E2 -17735.626} C_VEL
LIN {X 0,Y 268.627,Z 389.229,A -85,B 0,C 180,E1 -17738.274,E2 -17738.274} C_VEL
LIN {X 0,Y 269.158,Z 385.203,A -85,B 0,C 180,E1 -17740.532,E2 -17740.532} C_VEL
LIN {X 0,Y 270.141,Z 379.024,A -85,B 0,C 180,E1 -17743.158,E2 -17743.158} C_VEL
LIN {X 0,Y 271.501,Z 372.298,A -85,B 0,C 180,E1 -17745.387,E2 -17745.387} C_VEL
LIN {X 0,Y 273.063,Z 364.535,A -85,B 0,C 180,E1 -17747.456,E2 -17747.456} C_VEL
LIN {X 0,Y 274.644,Z 355.41,A -85,B 0,C 180,E1 -17749.431,E2 -17749.431} C_VEL
LIN {X 0,Y 276.708,Z 344.879,A -85,B 0,C 180,E1 -17751.219,E2 -17751.219} C_VEL
LIN {X 0,Y 277.388,Z 339.933,A -85,B 0,C 180,E1 -17751.945,E2 -17751.945} C_VEL
LIN {X 0,Y 277.073,Z 328.392,A -85,B 0,C 180,E1 -17753.516,E2 -17753.516} C_VEL
LIN {X 0,Y 276.171,Z 316.497,A -85,B 0,C 180,E1 -17754.851,E2 -17754.851} C_VEL
LIN {X 0,Y 274.279,Z 303.931,A -85,B 0,C 180,E1 -17756.027,E2 -17756.027} C_VEL
LIN {X 0,Y 271.339,Z 290.493,A -85,B 0,C 180,E1 -17757.065,E2 -17757.065} C_VEL
LIN {X 0,Y 270.68,Z 287.453,A -85,B 0,C 180,E1 -17757.273,E2 -17757.273} C_VEL
LIN {X 0,Y 271.692,Z 281.935,A -85,B 0,C 180,E1 -17761.155,E2 -17761.155} C_VEL
LIN {X 0,Y 272.948,Z 275.927,A -85,B 0,C 180,E1 -17765.405,E2 -17765.405} C_VEL
LIN {X 0,Y 273.285,Z 273.546,A -85,B 0,C 180,E1 -17767.134,E2 -17767.134} C_VEL
LIN {X 0,Y 272.936,Z 269.759,A -85,B 0,C 180,E1 -17770.072,E2 -17770.072} C_VEL
LIN {X 0,Y 272.012,Z 264.749,A -85,B 0,C 180,E1 -17774.236,E2 -17774.236} C_VEL
LIN {X 0,Y 271.323,Z 260.869,A -85,B 0,C 180,E1 -17777.664,E2 -17777.664} C_VEL
LIN {X 0,Y 270.586,Z 256.961,A -85,B 0,C 180,E1 -17781.438,E2 -17781.438} C_VEL
LIN {X 0,Y 270.236,Z 254.825,A -85,B 0,C 180,E1 -17783.729,E2 -17783.729} C_VEL
LIN {X 0,Y 270.204,Z 254.83,A -85,B 0,C 180,E1 -17786.893,E2 -17786.893} C_VEL
LIN {X 0,Y 270.185,Z 254.831,A -85,B 0,C 180,E1 -17790.381,E2 -17790.381} C_VEL
LIN {X 0,Y 270.198,Z 254.829,A -85,B 0,C 180,E1 -17793.757,E2 -17793.757} C_VEL
LIN {X 0,Y 270.189,Z 254.83,A -85,B 0,C 180,E1 -17797.035,E2 -17797.035} C_VEL
LIN {X 0,Y 270.292,Z 254.819,A -85,B 0,C 180,E1 -17800.244,E2 -17800.244} C_VEL
LIN {X 0,Y 270.407,Z 254.801,A -85,B 0,C 180,E1 -17804.936,E2 -17804.936} C_VEL
LIN {X 0,Y 270.413,Z 254.802,A -85,B 0,C 180,E1 -17809.518,E2 -17809.518} C_VEL
LIN {X 0,Y 270.585,Z 254.777,A -85,B 0,C 180,E1 -17812.538,E2 -17812.538} C_VEL
LIN {X 0,Y 270.79,Z 254.753,A -85,B 0,C 180,E1 -17818.513,E2 -17818.513} C_VEL
LIN {X 0,Y 270.775,Z 254.758,A -85,B 0,C 180,E1 -17821.487,E2 -17821.487} C_VEL
LIN {X 0,Y 270.585,Z 254.781,A -85,B 0,C 180,E1 -17827.462,E2 -17827.462} C_VEL
LIN {X 0,Y 270.414,Z 254.8,A -85,B 0,C 180,E1 -17830.482,E2 -17830.482} C_VEL
LIN {X 0,Y 270.372,Z 254.807,A -85,B 0,C 180,E1 -17835.067,E2 -17835.067} C_VEL
LIN {X 0,Y 270.261,Z 254.818,A -85,B 0,C 180,E1 -17839.759,E2 -17839.759} C_VEL
LIN {X 0,Y 270.227,Z 254.825,A -85,B 0,C 180,E1 -17844.59,E2 -17844.59} C_VEL
LIN {X 0,Y 270.202,Z 254.826,A -85,B 0,C 180,E1 -17847.917,E2 -17847.917} C_VEL
LIN {X 0,Y 270.176,Z 254.829,A -85,B 0,C 180,E1 -17851.349,E2 -17851.349} C_VEL
LIN {X 0,Y 270.205,Z 254.825,A -85,B 0,C 180,E1 -17854.905,E2 -17854.905} C_VEL
LIN {X 0,Y 270.2,Z 254.826,A -85,B 0,C 180,E1 -17858.71,E2 -17858.71} C_VEL
LIN {X 0,Y 270.175,Z 254.83,A -85,B 0,C 180,E1 -17862.558,E2 -17862.558} C_VEL
LIN {X 0,Y 270.168,Z 254.83,A -85,B 0,C 180,E1 -17866.751,E2 -17866.751} C_VEL
LIN {X 0,Y 270.176,Z 254.831,A -85,B 0,C 180,E1 -17869.434,E2 -17869.434} C_VEL
LIN {X 0,Y 270.096,Z 254.839,A -85,B 0,C 180,E1 -17873.239,E2 -17873.239} C_VEL
LIN {X 0,Y 269.952,Z 254.858,A -85,B 0,C 180,E1 -17875.057,E2 -17875.057} C_VEL
LIN {X 0,Y 269.909,Z 255.778,A -85,B 0,C 180,E1 -17876.851,E2 -17876.851} C_VEL
LIN {X 0,Y 269.781,Z 258.328,A -85,B 0,C 180,E1 -17880.332,E2 -17880.332} C_VEL
LIN {X 0,Y 269.727,Z 260.217,A -85,B 0,C 180,E1 -17882.752,E2 -17882.752} C_VEL
LIN {X 0,Y 271.64,Z 265.564,A -85,B 0,C 180,E1 -17883.21,E2 -17883.21} C_VEL
LIN {X 0,Y 275.64,Z 277.204,A -85,B 0,C 180,E1 -17884.374,E2 -17884.374} C_VEL
LIN {X 0,Y 278.573,Z 288.157,A -85,B 0,C 180,E1 -17885.622,E2 -17885.622} C_VEL
LIN {X 0,Y 280.577,Z 298.486,A -85,B 0,C 180,E1 -17886.959,E2 -17886.959} C_VEL
LIN {X 0,Y 280.527,Z 301.596,A -85,B 0,C 180,E1 -17887.344,E2 -17887.344} C_VEL
LIN {X 0,Y 278.84,Z 312.242,A -85,B 0,C 180,E1 -17888.76,E2 -17888.76} C_VEL
LIN {X 0,Y 277.276,Z 321.892,A -85,B 0,C 180,E1 -17890.376,E2 -17890.376} C_VEL
LIN {X 0,Y 275.476,Z 330.696,A -85,B 0,C 180,E1 -17892.173,E2 -17892.173} C_VEL
LIN {X 0,Y 273.981,Z 337.948,A -85,B 0,C 180,E1 -17893.993,E2 -17893.993} C_VEL
LIN {X 0,Y 272.494,Z 345.076,A -85,B 0,C 180,E1 -17896.198,E2 -17896.198} C_VEL
LIN {X 0,Y 271.305,Z 349.889,A -85,B 0,C 180,E1 -17898.039,E2 -17898.039} C_VEL
LIN {X 0,Y 270.298,Z 354.554,A -85,B 0,C 180,E1 -17900.27,E2 -17900.27} C_VEL
LIN {X 0,Y 269.622,Z 358.116,A -85,B 0,C 180,E1 -17902.511,E2 -17902.511} C_VEL
LIN {X 0,Y 269.227,Z 359.959,A -85,B 0,C 180,E1 -17904.006,E2 -17904.006} C_VEL
LIN {X 0,Y 268.918,Z 361.345,A -85,B 0,C 180,E1 -17905.503,E2 -17905.503} C_VEL
LIN {X 0,Y 268.604,Z 362.935,A -85,B 0,C 180,E1 -17908.5,E2 -17908.5} C_VEL
LIN {X 0,Y 268.582,Z 363.163,A -85,B 0,C 180,E1 -17910,E2 -17910} C_VEL
LIN {X 0,Y 268.602,Z 362.972,A -85,B 0,C 180,E1 -17911.499,E2 -17911.499} C_VEL
LIN {X 0,Y 268.904,Z 361.43,A -85,B 0,C 180,E1 -17914.497,E2 -17914.497} C_VEL
LIN {X 0,Y 269.207,Z 360.081,A -85,B 0,C 180,E1 -17915.994,E2 -17915.994} C_VEL
LIN {X 0,Y 269.748,Z 357.444,A -85,B 0,C 180,E1 -17918.087,E2 -17918.087} C_VEL
LIN {X 0,Y 270.577,Z 353.372,A -85,B 0,C 180,E1 -17920.476,E2 -17920.476} C_VEL
LIN {X 0,Y 271.694,Z 348.382,A -85,B 0,C 180,E1 -17922.701,E2 -17922.701} C_VEL
LIN {X 0,Y 273.07,Z 342.094,A -85,B 0,C 180,E1 -17924.914,E2 -17924.914} C_VEL
LIN {X 0,Y 274.768,Z 334.218,A -85,B 0,C 180,E1 -17927.106,E2 -17927.106} C_VEL
LIN {X 0,Y 276.869,Z 324.408,A -85,B 0,C 180,E1 -17929.268,E2 -17929.268} C_VEL
LIN {X 0,Y 278.536,Z 314.556,A -85,B 0,C 180,E1 -17930.999,E2 -17930.999} C_VEL
LIN {X 0,Y 280.255,Z 303.903,A -85,B 0,C 180,E1 -17932.484,E2 -17932.484} C_VEL
LIN {X 0,Y 280.768,Z 299.439,A -85,B 0,C 180,E1 -17933.024,E2 -17933.024} C_VEL
LIN {X 0,Y 278.599,Z 288.103,A -85,B 0,C 180,E1 -17934.503,E2 -17934.503} C_VEL
LIN {X 0,Y 275.253,Z 275.877,A -85,B 0,C 180,E1 -17935.889,E2 -17935.889} C_VEL
LIN {X 0,Y 270.854,Z 263.389,A -85,B 0,C 180,E1 -17937.103,E2 -17937.103} C_VEL
LIN {X 0,Y 269.686,Z 260.119,A -85,B 0,C 180,E1 -17937.401,E2 -17937.401} C_VEL
LIN {X 0,Y 269.831,Z 257.134,A -85,B 0,C 180,E1 -17941.394,E2 -17941.394} C_VEL
LIN {X 0,Y 269.925,Z 255.592,A -85,B 0,C 180,E1 -17943.573,E2 -17943.573} C_VEL
LIN {X 0,Y 269.946,Z 254.861,A -85,B 0,C 180,E1 -17944.943,E2 -17944.943} C_VEL
LIN {X 0,Y 270.168,Z 254.834,A -85,B 0,C 180,E1 -17948.702,E2 -17948.702} C_VEL
LIN {X 0,Y 270.173,Z 254.831,A -85,B 0,C 180,E1 -17952.558,E2 -17952.558} C_VEL
LIN {X 0,Y 270.167,Z 254.828,A -85,B 0,C 180,E1 -17956.751,E2 -17956.751} C_VEL
LIN {X 0,Y 270.176,Z 254.831,A -85,B 0,C 180,E1 -17959.434,E2 -17959.434} C_VEL
LIN {X 0,Y 270.229,Z 254.825,A -85,B 0,C 180,E1 -17963.73,E2 -17963.73} C_VEL
LIN {X 0,Y 270.203,Z 254.826,A -85,B 0,C 180,E1 -17966.892,E2 -17966.892} C_VEL
LIN {X 0,Y 270.184,Z 254.828,A -85,B 0,C 180,E1 -17970.381,E2 -17970.381} C_VEL
LIN {X 0,Y 270.204,Z 254.826,A -85,B 0,C 180,E1 -17973.757,E2 -17973.757} C_VEL
LIN {X 0,Y 270.204,Z 254.828,A -85,B 0,C 180,E1 -17977.036,E2 -17977.036} C_VEL
LIN {X 0,Y 270.259,Z 254.819,A -85,B 0,C 180,E1 -17980.241,E2 -17980.241} C_VEL
LIN {X 0,Y 270.37,Z 254.806,A -85,B 0,C 180,E1 -17984.933,E2 -17984.933} C_VEL
LIN {X 0,Y 270.444,Z 254.795,A -85,B 0,C 180,E1 -17989.519,E2 -17989.519} C_VEL
LIN {X 0,Y 270.613,Z 254.776,A -85,B 0,C 180,E1 -17992.539,E2 -17992.539} C_VEL
LIN {X 0,Y 270.774,Z 254.758,A -85,B 0,C 180,E1 -17998.513,E2 -17998.513} C_VEL
LIN {X 0,Y 270.788,Z 254.753,A -85,B 0,C 180,E1 -18001.487,E2 -18001.487} C_VEL
LIN {X 0,Y 270.587,Z 254.778,A -85,B 0,C 180,E1 -18007.462,E2 -18007.462} C_VEL
LIN {X 0,Y 270.411,Z 254.803,A -85,B 0,C 180,E1 -18010.482,E2 -18010.482} C_VEL
LIN {X 0,Y 270.405,Z 254.799,A -85,B 0,C 180,E1 -18015.065,E2 -18015.065} C_VEL
LIN {X 0,Y 270.385,Z 254.802,A -85,B 0,C 180,E1 -18015.547,E2 -18015.547} C_VEL
LIN {X 0,Y 269.698,Z 254.893,A -85,B 0,C 180,E1 -18016.789,E2 -18016.789} C_VEL
LIN {X 0,Y 266.798,Z 255.26,A -85,B 0,C 180,E1 -18018.811,E2 -18018.811} C_VEL
LIN {X 0,Y 264.321,Z 255.568,A -85,B 0,C 180,E1 -18020.455,E2 -18020.455} C_VEL
LIN {X 0,Y 263.227,Z 255.699,A -85,B 0,C 180,E1 -18021.73,E2 -18021.73} C_VEL
LIN {X 0,Y 263.121,Z 255.71,A -85,B 0,C 180,E1 -18022.163,E2 -18022.163} C_VEL
LIN {X 0,Y 263.128,Z 255.712,A -85,B 0,C 180,E1 -18025.3,E2 -18025.3} C_VEL
LIN {X 0,Y 263.134,Z 255.712,A -85,B 0,C 180,E1 -18028.735,E2 -18028.735} C_VEL
LIN {X 0,Y 263.129,Z 255.713,A -85,B 0,C 180,E1 -18032.289,E2 -18032.289} C_VEL
LIN {X 0,Y 263.184,Z 255.842,A -85,B 0,C 180,E1 -18035.743,E2 -18035.743} C_VEL
LIN {X 0,Y 263.848,Z 259.687,A -85,B 0,C 180,E1 -18039.738,E2 -18039.738} C_VEL
LIN {X 0,Y 264.617,Z 263.777,A -85,B 0,C 180,E1 -18043.673,E2 -18043.673} C_VEL
LIN {X 0,Y 265.498,Z 268.475,A -85,B 0,C 180,E1 -18047.833,E2 -18047.833} C_VEL
LIN {X 0,Y 266.099,Z 271.867,A -85,B 0,C 180,E1 -18050.664,E2 -18050.664} C_VEL
LIN {X 0,Y 266.235,Z 274.334,A -85,B 0,C 180,E1 -18052.616,E2 -18052.616} C_VEL
LIN {X 0,Y 265.746,Z 277.601,A -85,B 0,C 180,E1 -18055.069,E2 -18055.069} C_VEL
LIN {X 0,Y 264.417,Z 283.921,A -85,B 0,C 180,E1 -18059.668,E2 -18059.668} C_VEL
LIN {X 0,Y 263.806,Z 287.063,A -85,B 0,C 180,E1 -18061.929,E2 -18061.929} C_VEL
LIN {X 0,Y 267.126,Z 301.857,A -85,B 0,C 180,E1 -18063.084,E2 -18063.084} C_VEL
LIN {X 0,Y 269.234,Z 314.762,A -85,B 0,C 180,E1 -18064.322,E2 -18064.322} C_VEL
LIN {X 0,Y 270.292,Z 326.667,A -85,B 0,C 180,E1 -18065.675,E2 -18065.675} C_VEL
LIN {X 0,Y 270.626,Z 338.334,A -85,B 0,C 180,E1 -18067.276,E2 -18067.276} C_VEL
LIN {X 0,Y 270.312,Z 343.411,A -85,B 0,C 180,E1 -18068.053,E2 -18068.053} C_VEL
LIN {X 0,Y 268.317,Z 353.137,A -85,B 0,C 180,E1 -18069.693,E2 -18069.693} C_VEL
LIN {X 0,Y 266.378,Z 362.953,A -85,B 0,C 180,E1 -18071.77,E2 -18071.77} C_VEL
LIN {X 0,Y 264.848,Z 370.692,A -85,B 0,C 180,E1 -18073.822,E2 -18073.822} C_VEL
LIN {X 0,Y 263.459,Z 377.635,A -85,B 0,C 180,E1 -18076.109,E2 -18076.109} C_VEL
LIN {X 0,Y 262.38,Z 383.206,A -85,B 0,C 180,E1 -18078.411,E2 -18078.411} C_VEL
LIN {X 0,Y 261.736,Z 387.59,A -85,B 0,C 180,E1 -18080.729,E2 -18080.729} C_VEL
LIN {X 0,Y 261.474,Z 389.916,A -85,B 0,C 180,E1 -18082.277,E2 -18082.277} C_VEL
LIN {X 0,Y 261.328,Z 392.27,A -85,B 0,C 180,E1 -18084.302,E2 -18084.302} C_VEL
LIN {X 0,Y 261.272,Z 394.24,A -85,B 0,C 180,E1 -18086.916,E2 -18086.916} C_VEL
LIN {X 0,Y 261.255,Z 394.858,A -85,B 0,C 180,E1 -18088.459,E2 -18088.459} C_VEL
LIN {X 0,Y 261.34,Z 395.08,A -85,B 0,C 180,E1 -18090,E2 -18090} C_VEL
LIN {X 0,Y 261.255,Z 394.852,A -85,B 0,C 180,E1 -18091.542,E2 -18091.542} C_VEL
LIN {X 0,Y 261.271,Z 394.23,A -85,B 0,C 180,E1 -18093.084,E2 -18093.084} C_VEL
LIN {X 0,Y 261.262,Z 392.393,A -85,B 0,C 180,E1 -18095.551,E2 -18095.551} C_VEL
LIN {X 0,Y 261.572,Z 388.799,A -85,B 0,C 180,E1 -18098.498,E2 -18098.498} C_VEL
LIN {X 0,Y 262.125,Z 384.771,A -85,B 0,C 180,E1 -18100.818,E2 -18100.818} C_VEL
LIN {X 0,Y 263.209,Z 378.594,A -85,B 0,C 180,E1 -18103.512,E2 -18103.512} C_VEL
LIN {X 0,Y 264.583,Z 371.864,A -85,B 0,C 180,E1 -18105.799,E2 -18105.799} C_VEL
LIN {X 0,Y 266.306,Z 363.771,A -85,B 0,C 180,E1 -18108.001,E2 -18108.001} C_VEL
LIN {X 0,Y 267.922,Z 354.977,A -85,B 0,C 180,E1 -18109.939,E2 -18109.939} C_VEL
LIN {X 0,Y 270.082,Z 344.446,A -85,B 0,C 180,E1 -18111.766,E2 -18111.766} C_VEL
LIN {X 0,Y 270.599,Z 340.8,A -85,B 0,C 180,E1 -18112.324,E2 -18112.324} C_VEL
LIN {X 0,Y 270.358,Z 329.091,A -85,B 0,C 180,E1 -18113.992,E2 -18113.992} C_VEL
LIN {X 0,Y 269.571,Z 317.975,A -85,B 0,C 180,E1 -18115.312,E2 -18115.312} C_VEL
LIN {X 0,Y 267.963,Z 306.442,A -85,B 0,C 180,E1 -18116.479,E2 -18116.479} C_VEL
LIN {X 0,Y 265.346,Z 293.636,A -85,B 0,C 180,E1 -18117.561,E2 -18117.561} C_VEL
LIN {X 0,Y 263.786,Z 287.017,A -85,B 0,C 180,E1 -18118.049,E2 -18118.049} C_VEL
LIN {X 0,Y 264.892,Z 281.505,A -85,B 0,C 180,E1 -18122.049,E2 -18122.049} C_VEL
LIN {X 0,Y 265.924,Z 276.709,A -85,B 0,C 180,E1 -18125.552,E2 -18125.552} C_VEL
LIN {X 0,Y 266.26,Z 273.952,A -85,B 0,C 180,E1 -18127.64,E2 -18127.64} C_VEL
LIN {X 0,Y 265.971,Z 271.027,A -85,B 0,C 180,E1 -18129.978,E2 -18129.978} C_VEL
LIN {X 0,Y 265.037,Z 265.995,A -85,B 0,C 180,E1 -18134.278,E2 -18134.278} C_VEL
LIN {X 0,Y 264.243,Z 261.63,A -85,B 0,C 180,E1 -18138.324,E2 -18138.324} C_VEL
LIN {X 0,Y 263.382,Z 256.772,A -85,B 0,C 180,E1 -18143.18,E2 -18143.18} C_VEL
LIN {X 0,Y 263.168,Z 255.71,A -85,B 0,C 180,E1 -18144.49,E2 -18144.49} C_VEL
LIN {X 0,Y 263.132,Z 255.709,A -85,B 0,C 180,E1 -18148.727,E2 -18148.727} C_VEL
LIN {X 0,Y 263.14,Z 255.708,A -85,B 0,C 180,E1 -18152.997,E2 -18152.997} C_VEL
LIN {X 0,Y 263.122,Z 255.712,A -85,B 0,C 180,E1 -18156.381,E2 -18156.381} C_VEL
LIN {X 0,Y 263.252,Z 255.695,A -85,B 0,C 180,E1 -18159.692,E2 -18159.692} C_VEL
LIN {X 0,Y 263.355,Z 255.68,A -85,B 0,C 180,E1 -18164.522,E2 -18164.522} C_VEL
LIN {X 0,Y 263.356,Z 255.68,A -85,B 0,C 180,E1 -18169.234,E2 -18169.234} C_VEL
LIN {X 0,Y 263.545,Z 255.655,A -85,B 0,C 180,E1 -18172.338,E2 -18172.338} C_VEL
LIN {X 0,Y 263.754,Z 255.629,A -85,B 0,C 180,E1 -18178.473,E2 -18178.473} C_VEL
LIN {X 0,Y 263.739,Z 255.635,A -85,B 0,C 180,E1 -18181.527,E2 -18181.527} C_VEL
LIN {X 0,Y 263.545,Z 255.656,A -85,B 0,C 180,E1 -18187.663,E2 -18187.663} C_VEL
LIN {X 0,Y 263.353,Z 255.681,A -85,B 0,C 180,E1 -18190.767,E2 -18190.767} C_VEL
LIN {X 0,Y 263.314,Z 255.685,A -85,B 0,C 180,E1 -18195.48,E2 -18195.48} C_VEL
LIN {X 0,Y 263.241,Z 255.694,A -85,B 0,C 180,E1 -18200.309,E2 -18200.309} C_VEL
LIN {X 0,Y 263.171,Z 255.702,A -85,B 0,C 180,E1 -18205.295,E2 -18205.295} C_VEL
LIN {X 0,Y 263.137,Z 255.708,A -85,B 0,C 180,E1 -18208.735,E2 -18208.735} C_VEL
LIN {X 0,Y 263.131,Z 255.71,A -85,B 0,C 180,E1 -18212.289,E2 -18212.289} C_VEL
LIN {X 0,Y 263.188,Z 255.701,A -85,B 0,C 180,E1 -18216.764,E2 -18216.764} C_VEL
LIN {X 0,Y 263.127,Z 255.709,A -85,B 0,C 180,E1 -18221.593,E2 -18221.593} C_VEL
LIN {X 0,Y 263.125,Z 255.711,A -85,B 0,C 180,E1 -18226.016,E2 -18226.016} C_VEL
LIN {X 0,Y 263.099,Z 255.713,A -85,B 0,C 180,E1 -18230.126,E2 -18230.126} C_VEL
LIN {X 0,Y 262.997,Z 255.724,A -85,B 0,C 180,E1 -18233.991,E2 -18233.991} C_VEL
LIN {X 0,Y 262.904,Z 256.301,A -85,B 0,C 180,E1 -18235.966,E2 -18235.966} C_VEL
LIN {X 0,Y 262.8,Z 258.759,A -85,B 0,C 180,E1 -18239.461,E2 -18239.461} C_VEL
LIN {X 0,Y 262.745,Z 260.833,A -85,B 0,C 180,E1 -18241.97,E2 -18241.97} C_VEL
LIN {X 0,Y 267.555,Z 273.958,A -85,B 0,C 180,E1 -18243.265,E2 -18243.265} C_VEL
LIN {X 0,Y 271.008,Z 285.625,A -85,B 0,C 180,E1 -18244.597,E2 -18244.597} C_VEL
LIN {X 0,Y 273.239,Z 295.695,A -85,B 0,C 180,E1 -18245.9,E2 -18245.9} C_VEL
LIN {X 0,Y 274.018,Z 300.48,A -85,B 0,C 180,E1 -18246.575,E2 -18246.575} C_VEL
LIN {X 0,Y 272.893,Z 308.92,A -85,B 0,C 180,E1 -18247.675,E2 -18247.675} C_VEL
LIN {X 0,Y 271.173,Z 319.36,A -85,B 0,C 180,E1 -18249.329,E2 -18249.329} C_VEL
LIN {X 0,Y 269.492,Z 327.825,A -85,B 0,C 180,E1 -18250.974,E2 -18250.974} C_VEL
LIN {X 0,Y 267.834,Z 335.653,A -85,B 0,C 180,E1 -18252.83,E2 -18252.83} C_VEL
LIN {X 0,Y 266.047,Z 343.302,A -85,B 0,C 180,E1 -18255.074,E2 -18255.074} C_VEL
LIN {X 0,Y 264.846,Z 348.518,A -85,B 0,C 180,E1 -18256.964,E2 -18256.964} C_VEL
LIN {X 0,Y 263.641,Z 353.575,A -85,B 0,C 180,E1 -18259.245,E2 -18259.245} C_VEL
LIN {X 0,Y 262.718,Z 357.861,A -85,B 0,C 180,E1 -18261.808,E2 -18261.808} C_VEL
LIN {X 0,Y 262.198,Z 360.386,A -85,B 0,C 180,E1 -18263.845,E2 -18263.845} C_VEL
LIN {X 0,Y 261.863,Z 361.772,A -85,B 0,C 180,E1 -18265.382,E2 -18265.382} C_VEL
LIN {X 0,Y 261.519,Z 363.363,A -85,B 0,C 180,E1 -18268.46,E2 -18268.46} C_VEL
LIN {X 0,Y 261.495,Z 363.59,A -85,B 0,C 180,E1 -18270,E2 -18270} C_VEL
LIN {X 0,Y 261.517,Z 363.399,A -85,B 0,C 180,E1 -18271.54,E2 -18271.54} C_VEL
LIN {X 0,Y 261.849,Z 361.856,A -85,B 0,C 180,E1 -18274.618,E2 -18274.618} C_VEL
LIN {X 0,Y 262.176,Z 360.506,A -85,B 0,C 180,E1 -18276.155,E2 -18276.155} C_VEL
LIN {X 0,Y 262.667,Z 358.129,A -85,B 0,C 180,E1 -18278.115,E2 -18278.115} C_VEL
LIN {X 0,Y 263.612,Z 353.797,A -85,B 0,C 180,E1 -18280.756,E2 -18280.756} C_VEL
LIN {X 0,Y 264.79,Z 348.807,A -85,B 0,C 180,E1 -18283.038,E2 -18283.038} C_VEL
LIN {X 0,Y 266.233,Z 342.518,A -85,B 0,C 180,E1 -18285.306,E2 -18285.306} C_VEL
LIN {X 0,Y 268.015,Z 334.641,A -85,B 0,C 180,E1 -18287.551,E2 -18287.551} C_VEL
LIN {X 0,Y 270.205,Z 324.83,A -85,B 0,C 180,E1 -18289.763,E2 -18289.763} C_VEL
LIN {X 0,Y 271.843,Z 315.498,A -85,B 0,C 180,E1 -18291.453,E2 -18291.453} C_VEL
LIN {X 0,Y 273.475,Z 305.744,A -85,B 0,C 180,E1 -18292.873,E2 -18292.873} C_VEL
LIN {X 0,Y 274.15,Z 301.426,A -85,B 0,C 180,E1 -18293.413,E2 -18293.413} C_VEL
LIN {X 0,Y 272.27,Z 290.749,A -85,B 0,C 180,E1 -18294.879,E2 -18294.879} C_VEL
LIN {X 0,Y 269.04,Z 278.437,A -85,B 0,C 180,E1 -18296.365,E2 -18296.365} C_VEL
LIN {X 0,Y 264.911,Z 266.586,A -85,B 0,C 180,E1 -18297.625,E2 -18297.625} C_VEL
LIN {X 0,Y 262.787,Z 261.264,A -85,B 0,C 180,E1 -18298.134,E2 -18298.134} C_VEL
LIN {X 0,Y 262.684,Z 260.582,A -85,B 0,C 180,E1 -18298.178,E2 -18298.178} C_VEL
LIN {X 0,Y 262.853,Z 257.573,A -85,B 0,C 180,E1 -18302.327,E2 -18302.327} C_VEL
LIN {X 0,Y 262.903,Z 256.324,A -85,B 0,C 180,E1 -18304.151,E2 -18304.151} C_VEL
LIN {X 0,Y 263.05,Z 255.723,A -85,B 0,C 180,E1 -18306.724,E2 -18306.724} C_VEL
LIN {X 0,Y 263.098,Z 255.714,A -85,B 0,C 180,E1 -18309.874,E2 -18309.874} C_VEL
LIN {X 0,Y 263.124,Z 255.708,A -85,B 0,C 180,E1 -18313.984,E2 -18313.984} C_VEL
LIN {X 0,Y 263.126,Z 255.709,A -85,B 0,C 180,E1 -18318.406,E2 -18318.406} C_VEL
LIN {X 0,Y 263.186,Z 255.701,A -85,B 0,C 180,E1 -18323.236,E2 -18323.236} C_VEL
LIN {X 0,Y 263.13,Z 255.709,A -85,B 0,C 180,E1 -18327.711,E2 -18327.711} C_VEL
LIN {X 0,Y 263.149,Z 255.706,A -85,B 0,C 180,E1 -18331.805,E2 -18331.805} C_VEL
LIN {X 0,Y 263.191,Z 255.7,A -85,B 0,C 180,E1 -18335.218,E2 -18335.218} C_VEL
LIN {X 0,Y 263.239,Z 255.695,A -85,B 0,C 180,E1 -18339.691,E2 -18339.691} C_VEL
LIN {X 0,Y 263.312,Z 255.685,A -85,B 0,C 180,E1 -18344.52,E2 -18344.52} C_VEL
LIN {X 0,Y 263.376,Z 255.677,A -85,B 0,C 180,E1 -18349.234,E2 -18349.234} C_VEL
LIN {X 0,Y 263.575,Z 255.652,A -85,B 0,C 180,E1 -18352.338,E2 -18352.338} C_VEL
LIN {X 0,Y 263.738,Z 255.635,A -85,B 0,C 180,E1 -18358.473,E2 -18358.473} C_VEL
LIN {X 0,Y 263.752,Z 255.63,A -85,B 0,C 180,E1 -18361.527,E2 -18361.527} C_VEL
LIN {X 0,Y 263.546,Z 255.655,A -85,B 0,C 180,E1 -18367.662,E2 -18367.662} C_VEL
LIN {X 0,Y 263.354,Z 255.68,A -85,B 0,C 180,E1 -18370.766,E2 -18370.766} C_VEL
LIN {X 0,Y 263.351,Z 255.678,A -85,B 0,C 180,E1 -18375.538,E2 -18375.538} C_VEL
LIN {X 0,Y 263.251,Z 255.695,A -85,B 0,C 180,E1 -18380.308,E2 -18380.308} C_VEL
LIN {X 0,Y 263.121,Z 255.71,A -85,B 0,C 180,E1 -18382.163,E2 -18382.163} C_VEL
LIN {X 0,Y 262.419,Z 255.799,A -85,B 0,C 180,E1 -18383.44,E2 -18383.44} C_VEL
LIN {X 0,Y 259.594,Z 256.152,A -85,B 0,C 180,E1 -18385.523,E2 -18385.523} C_VEL
LIN {X 0,Y 257.207,Z 256.45,A -85,B 0,C 180,E1 -18387.217,E2 -18387.217} C_VEL
LIN {X 0,Y 256.164,Z 256.581,A -85,B 0,C 180,E1 -18388.528,E2 -18388.528} C_VEL
LIN {X 0,Y 256.067,Z 256.592,A -85,B 0,C 180,E1 -18388.973,E2 -18388.973} C_VEL
LIN {X 0,Y 256.067,Z 256.592,A -85,B 0,C 180,E1 -18393.293,E2 -18393.293} C_VEL
LIN {X 0,Y 256.108,Z 256.593,A -85,B 0,C 180,E1 -18394.818,E2 -18394.818} C_VEL
LIN {X 0,Y 256.77,Z 260.431,A -85,B 0,C 180,E1 -18399.015,E2 -18399.015} C_VEL
LIN {X 0,Y 257.51,Z 264.482,A -85,B 0,C 180,E1 -18403.024,E2 -18403.024} C_VEL
LIN {X 0,Y 258.39,Z 269.046,A -85,B 0,C 180,E1 -18407.255,E2 -18407.255} C_VEL
LIN {X 0,Y 259.069,Z 272.754,A -85,B 0,C 180,E1 -18410.467,E2 -18410.467} C_VEL
LIN {X 0,Y 259.113,Z 276.339,A -85,B 0,C 180,E1 -18413.365,E2 -18413.365} C_VEL
LIN {X 0,Y 258.096,Z 281.125,A -85,B 0,C 180,E1 -18417.002,E2 -18417.002} C_VEL
LIN {X 0,Y 256.974,Z 286.793,A -85,B 0,C 180,E1 -18421.141,E2 -18421.141} C_VEL
LIN {X 0,Y 260.096,Z 300.376,A -85,B 0,C 180,E1 -18422.223,E2 -18422.223} C_VEL
LIN {X 0,Y 262.323,Z 313.165,A -85,B 0,C 180,E1 -18423.486,E2 -18423.486} C_VEL
LIN {X 0,Y 263.518,Z 325.708,A -85,B 0,C 180,E1 -18424.947,E2 -18424.947} C_VEL
LIN {X 0,Y 263.838,Z 336.565,A -85,B 0,C 180,E1 -18426.449,E2 -18426.449} C_VEL
LIN {X 0,Y 263.722,Z 342.986,A -85,B 0,C 180,E1 -18427.475,E2 -18427.475} C_VEL
LIN {X 0,Y 261.645,Z 352.711,A -85,B 0,C 180,E1 -18429.151,E2 -18429.151} C_VEL
LIN {X 0,Y 259.786,Z 361.591,A -85,B 0,C 180,E1 -18431.057,E2 -18431.057} C_VEL
LIN {X 0,Y 258.342,Z 368.94,A -85,B 0,C 180,E1 -18432.996,E2 -18432.996} C_VEL
LIN {X 0,Y 256.738,Z 376.174,A -85,B 0,C 180,E1 -18435.333,E2 -18435.333} C_VEL
LIN {X 0,Y 255.659,Z 381.063,A -85,B 0,C 180,E1 -18437.296,E2 -18437.296} C_VEL
LIN {X 0,Y 254.875,Z 385.834,A -85,B 0,C 180,E1 -18439.675,E2 -18439.675} C_VEL
LIN {X 0,Y 254.401,Z 389.487,A -85,B 0,C 180,E1 -18442.061,E2 -18442.061} C_VEL
LIN {X 0,Y 254.229,Z 392.067,A -85,B 0,C 180,E1 -18444.384,E2 -18444.384} C_VEL
LIN {X 0,Y 254.18,Z 393.813,A -85,B 0,C 180,E1 -18446.83,E2 -18446.83} C_VEL
LIN {X 0,Y 254.18,Z 394.432,A -85,B 0,C 180,E1 -18448.416,E2 -18448.416} C_VEL
LIN {X 0,Y 254.258,Z 394.654,A -85,B 0,C 180,E1 -18450,E2 -18450} C_VEL
LIN {X 0,Y 254.18,Z 394.425,A -85,B 0,C 180,E1 -18451.585,E2 -18451.585} C_VEL
LIN {X 0,Y 254.179,Z 393.802,A -85,B 0,C 180,E1 -18453.17,E2 -18453.17} C_VEL
LIN {X 0,Y 254.185,Z 392.143,A -85,B 0,C 180,E1 -18455.515,E2 -18455.515} C_VEL
LIN {X 0,Y 254.538,Z 388.37,A -85,B 0,C 180,E1 -18458.735,E2 -18458.735} C_VEL
LIN {X 0,Y 255.111,Z 384.34,A -85,B 0,C 180,E1 -18461.119,E2 -18461.119} C_VEL
LIN {X 0,Y 256.294,Z 378.163,A -85,B 0,C 180,E1 -18463.883,E2 -18463.883} C_VEL
LIN {X 0,Y 257.708,Z 371.431,A -85,B 0,C 180,E1 -18466.232,E2 -18466.232} C_VEL
LIN {X 0,Y 259.375,Z 364.031,A -85,B 0,C 180,E1 -18468.31,E2 -18468.31} C_VEL
LIN {X 0,Y 261.224,Z 354.544,A -85,B 0,C 180,E1 -18470.473,E2 -18470.473} C_VEL
LIN {X 0,Y 263.463,Z 344.012,A -85,B 0,C 180,E1 -18472.342,E2 -18472.342} C_VEL
LIN {X 0,Y 263.852,Z 339.042,A -85,B 0,C 180,E1 -18473.134,E2 -18473.134} C_VEL
LIN {X 0,Y 263.556,Z 327.577,A -85,B 0,C 180,E1 -18474.79,E2 -18474.79} C_VEL
LIN {X 0,Y 262.739,Z 316.852,A -85,B 0,C 180,E1 -18476.088,E2 -18476.088} C_VEL
LIN {X 0,Y 260.873,Z 304.151,A -85,B 0,C 180,E1 -18477.393,E2 -18477.393} C_VEL
LIN {X 0,Y 257.865,Z 290.802,A -85,B 0,C 180,E1 -18478.544,E2 -18478.544} C_VEL
LIN {X 0,Y 256.905,Z 286.578,A -85,B 0,C 180,E1 -18478.844,E2 -18478.844} C_VEL
LIN {X 0,Y 258.092,Z 281.077,A -85,B 0,C 180,E1 -18482.999,E2 -18482.999} C_VEL
LIN {X 0,Y 259.119,Z 276.292,A -85,B 0,C 180,E1 -18486.634,E2 -18486.634} C_VEL
LIN {X 0,Y 259.063,Z 272.705,A -85,B 0,C 180,E1 -18489.534,E2 -18489.534} C_VEL
LIN {X 0,Y 258.147,Z 267.735,A -85,B 0,C 180,E1 -18493.883,E2 -18493.883} C_VEL
LIN {X 0,Y 257.414,Z 263.882,A -85,B 0,C 180,E1 -18497.491,E2 -18497.491} C_VEL
LIN {X 0,Y 256.753,Z 260.377,A -85,B 0,C 180,E1 -18500.981,E2 -18500.981} C_VEL
LIN {X 0,Y 256.124,Z 256.619,A -85,B 0,C 180,E1 -18505.092,E2 -18505.092} C_VEL
LIN {X 0,Y 256.085,Z 256.585,A -85,B 0,C 180,E1 -18508.571,E2 -18508.571} C_VEL
LIN {X 0,Y 256.094,Z 256.587,A -85,B 0,C 180,E1 -18512.191,E2 -18512.191} C_VEL
LIN {X 0,Y 256.091,Z 256.588,A -85,B 0,C 180,E1 -18515.691,E2 -18515.691} C_VEL
LIN {X 0,Y 256.152,Z 256.579,A -85,B 0,C 180,E1 -18519.104,E2 -18519.104} C_VEL
LIN {X 0,Y 256.304,Z 256.56,A -85,B 0,C 180,E1 -18524.085,E2 -18524.085} C_VEL
LIN {X 0,Y 256.299,Z 256.558,A -85,B 0,C 180,E1 -18528.934,E2 -18528.934} C_VEL
LIN {X 0,Y 256.505,Z 256.533,A -85,B 0,C 180,E1 -18532.126,E2 -18532.126} C_VEL
LIN {X 0,Y 256.501,Z 256.534,A -85,B 0,C 180,E1 -18536.859,E2 -18536.859} C_VEL
LIN {X 0,Y 256.717,Z 256.506,A -85,B 0,C 180,E1 -18538.431,E2 -18538.431} C_VEL
LIN {X 0,Y 256.702,Z 256.511,A -85,B 0,C 180,E1 -18541.569,E2 -18541.569} C_VEL
LIN {X 0,Y 256.463,Z 256.534,A -85,B 0,C 180,E1 -18546.719,E2 -18546.719} C_VEL
LIN {X 0,Y 256.43,Z 256.544,A -85,B 0,C 180,E1 -18549.465,E2 -18549.465} C_VEL
LIN {X 0,Y 256.236,Z 256.566,A -85,B 0,C 180,E1 -18554.291,E2 -18554.291} C_VEL
LIN {X 0,Y 256.177,Z 256.572,A -85,B 0,C 180,E1 -18557.564,E2 -18557.564} C_VEL
LIN {X 0,Y 256.145,Z 256.579,A -85,B 0,C 180,E1 -18561.111,E2 -18561.111} C_VEL
LIN {X 0,Y 256.136,Z 256.579,A -85,B 0,C 180,E1 -18565.112,E2 -18565.112} C_VEL
LIN {X 0,Y 256.058,Z 256.588,A -85,B 0,C 180,E1 -18569.607,E2 -18569.607} C_VEL
LIN {X 0,Y 256.069,Z 256.586,A -85,B 0,C 180,E1 -18573.293,E2 -18573.293} C_VEL
LIN {X 0,Y 256.119,Z 256.58,A -85,B 0,C 180,E1 -18577.271,E2 -18577.271} C_VEL
LIN {X 0,Y 256.058,Z 256.589,A -85,B 0,C 180,E1 -18581.203,E2 -18581.203} C_VEL
LIN {X 0,Y 256.06,Z 256.587,A -85,B 0,C 180,E1 -18585.53,E2 -18585.53} C_VEL
LIN {X 0,Y 256.055,Z 256.59,A -85,B 0,C 180,E1 -18588.796,E2 -18588.796} C_VEL
LIN {X 0,Y 255.997,Z 256.595,A -85,B 0,C 180,E1 -18592.844,E2 -18592.844} C_VEL
LIN {X 0,Y 255.871,Z 256.661,A -85,B 0,C 180,E1 -18594.773,E2 -18594.773} C_VEL
LIN {X 0,Y 255.796,Z 259.215,A -85,B 0,C 180,E1 -18598.531,E2 -18598.531} C_VEL
LIN {X 0,Y 255.754,Z 261.25,A -85,B 0,C 180,E1 -18601.129,E2 -18601.129} C_VEL
LIN {X 0,Y 256.847,Z 264.291,A -85,B 0,C 180,E1 -18601.416,E2 -18601.416} C_VEL
LIN {X 0,Y 260.983,Z 275.374,A -85,B 0,C 180,E1 -18602.606,E2 -18602.606} C_VEL
LIN {X 0,Y 264.475,Z 287.194,A -85,B 0,C 180,E1 -18604.03,E2 -18604.03} C_VEL
LIN {X 0,Y 266.862,Z 298.378,A -85,B 0,C 180,E1 -18605.565,E2 -18605.565} C_VEL
LIN {X 0,Y 267.452,Z 302.716,A -85,B 0,C 180,E1 -18606.205,E2 -18606.205} C_VEL
LIN {X 0,Y 265.634,Z 313.466,A -85,B 0,C 180,E1 -18607.712,E2 -18607.712} C_VEL
LIN {X 0,Y 263.959,Z 322.868,A -85,B 0,C 180,E1 -18609.366,E2 -18609.366} C_VEL
LIN {X 0,Y 262.037,Z 331.554,A -85,B 0,C 180,E1 -18611.225,E2 -18611.225} C_VEL
LIN {X 0,Y 260.092,Z 340.128,A -85,B 0,C 180,E1 -18613.517,E2 -18613.517} C_VEL
LIN {X 0,Y 258.497,Z 346.956,A -85,B 0,C 180,E1 -18615.836,E2 -18615.836} C_VEL
LIN {X 0,Y 257.053,Z 352.427,A -85,B 0,C 180,E1 -18618.167,E2 -18618.167} C_VEL
LIN {X 0,Y 256.053,Z 356.71,A -85,B 0,C 180,E1 -18620.521,E2 -18620.521} C_VEL
LIN {X 0,Y 255.566,Z 358.972,A -85,B 0,C 180,E1 -18622.097,E2 -18622.097} C_VEL
LIN {X 0,Y 255.171,Z 360.812,A -85,B 0,C 180,E1 -18623.675,E2 -18623.675} C_VEL
LIN {X 0,Y 254.813,Z 362.199,A -85,B 0,C 180,E1 -18625.253,E2 -18625.253} C_VEL
LIN {X 0,Y 254.436,Z 363.79,A -85,B 0,C 180,E1 -18628.417,E2 -18628.417} C_VEL
LIN {X 0,Y 254.409,Z 364.017,A -85,B 0,C 180,E1 -18630,E2 -18630} C_VEL
LIN {X 0,Y 254.435,Z 363.825,A -85,B 0,C 180,E1 -18631.583,E2 -18631.583} C_VEL
LIN {X 0,Y 254.799,Z 362.281,A -85,B 0,C 180,E1 -18634.746,E2 -18634.746} C_VEL
LIN {X 0,Y 255.148,Z 360.931,A -85,B 0,C 180,E1 -18636.325,E2 -18636.325} C_VEL
LIN {X 0,Y 255.609,Z 358.768,A -85,B 0,C 180,E1 -18638.179,E2 -18638.179} C_VEL
LIN {X 0,Y 256.637,Z 354.224,A -85,B 0,C 180,E1 -18641.052,E2 -18641.052} C_VEL
LIN {X 0,Y 257.887,Z 349.232,A -85,B 0,C 180,E1 -18643.394,E2 -18643.394} C_VEL
LIN {X 0,Y 259.417,Z 342.942,A -85,B 0,C 180,E1 -18645.719,E2 -18645.719} C_VEL
LIN {X 0,Y 261.283,Z 335.065,A -85,B 0,C 180,E1 -18648.019,E2 -18648.019} C_VEL
LIN {X 0,Y 263.565,Z 325.253,A -85,B 0,C 180,E1 -18650.282,E2 -18650.282} C_VEL
LIN {X 0,Y 265.354,Z 315.402,A -85,B 0,C 180,E1 -18652.096,E2 -18652.096} C_VEL
LIN {X 0,Y 267.236,Z 304.768,A -85,B 0,C 180,E1 -18653.641,E2 -18653.641} C_VEL
LIN {X 0,Y 267.442,Z 301.912,A -85,B 0,C 180,E1 -18654.03,E2 -18654.03} C_VEL
LIN {X 0,Y 265.475,Z 291.189,A -85,B 0,C 180,E1 -18655.562,E2 -18655.562} C_VEL
LIN {X 0,Y 262.766,Z 280.848,A -85,B 0,C 180,E1 -18656.878,E2 -18656.878} C_VEL
LIN {X 0,Y 258.689,Z 268.995,A -85,B 0,C 180,E1 -18658.227,E2 -18658.227} C_VEL
LIN {X 0,Y 255.791,Z 261.64,A -85,B 0,C 180,E1 -18658.979,E2 -18658.979} C_VEL
LIN {X 0,Y 255.685,Z 261.028,A -85,B 0,C 180,E1 -18659.034,E2 -18659.034} C_VEL
LIN {X 0,Y 255.808,Z 259.203,A -85,B 0,C 180,E1 -18661.604,E2 -18661.604} C_VEL
LIN {X 0,Y 255.869,Z 256.766,A -85,B 0,C 180,E1 -18665.227,E2 -18665.227} C_VEL
LIN {X 0,Y 256.009,Z 256.6,A -85,B 0,C 180,E1 -18667.239,E2 -18667.239} C_VEL
LIN {X 0,Y 256.054,Z 256.59,A -85,B 0,C 180,E1 -18671.204,E2 -18671.204} C_VEL
LIN {X 0,Y 256.059,Z 256.59,A -85,B 0,C 180,E1 -18675.53,E2 -18675.53} C_VEL
LIN {X 0,Y 256.056,Z 256.588,A -85,B 0,C 180,E1 -18678.797,E2 -18678.797} C_VEL
LIN {X 0,Y 256.134,Z 256.579,A -85,B 0,C 180,E1 -18682.868,E2 -18682.868} C_VEL
LIN {X 0,Y 256.067,Z 256.587,A -85,B 0,C 180,E1 -18686.707,E2 -18686.707} C_VEL
LIN {X 0,Y 256.056,Z 256.588,A -85,B 0,C 180,E1 -18690.393,E2 -18690.393} C_VEL
LIN {X 0,Y 256.134,Z 256.578,A -85,B 0,C 180,E1 -18694.888,E2 -18694.888} C_VEL
LIN {X 0,Y 256.15,Z 256.577,A -85,B 0,C 180,E1 -18699.103,E2 -18699.103} C_VEL
LIN {X 0,Y 256.246,Z 256.564,A -85,B 0,C 180,E1 -18704.081,E2 -18704.081} C_VEL
LIN {X 0,Y 256.291,Z 256.56,A -85,B 0,C 180,E1 -18707.328,E2 -18707.328} C_VEL
LIN {X 0,Y 256.499,Z 256.534,A -85,B 0,C 180,E1 -18710.538,E2 -18710.538} C_VEL
LIN {X 0,Y 256.487,Z 256.534,A -85,B 0,C 180,E1 -18713.707,E2 -18713.707} C_VEL
LIN {X 0,Y 256.7,Z 256.511,A -85,B 0,C 180,E1 -18718.431,E2 -18718.431} C_VEL
LIN {X 0,Y 256.715,Z 256.507,A -85,B 0,C 180,E1 -18721.569,E2 -18721.569} C_VEL
LIN {X 0,Y 256.477,Z 256.537,A -85,B 0,C 180,E1 -18726.293,E2 -18726.293} C_VEL
LIN {X 0,Y 256.428,Z 256.541,A -85,B 0,C 180,E1 -18729.465,E2 -18729.465} C_VEL
LIN {X 0,Y 256.257,Z 256.564,A -85,B 0,C 180,E1 -18734.29,E2 -18734.29} C_VEL
LIN {X 0,Y 256.212,Z 256.57,A -85,B 0,C 180,E1 -18737.562,E2 -18737.562} C_VEL
LIN {X 0,Y 256.144,Z 256.579,A -85,B 0,C 180,E1 -18741.111,E2 -18741.111} C_VEL
LIN {X 0,Y 256.087,Z 256.588,A -85,B 0,C 180,E1 -18745.09,E2 -18745.09} C_VEL
LIN {X 0,Y 256.067,Z 256.592,A -85,B 0,C 180,E1 -18748.973,E2 -18748.973} C_VEL
LIN {X 0,Y 255.371,Z 256.681,A -85,B 0,C 180,E1 -18750.286,E2 -18750.286} C_VEL
LIN {X 0,Y 252.556,Z 257.099,A -85,B 0,C 180,E1 -18752.427,E2 -18752.427} C_VEL
LIN {X 0,Y 250.261,Z 257.873,A -85,B 0,C 180,E1 -18754.161,E2 -18754.161} C_VEL
LIN {X 0,Y 249.372,Z 258.777,A -85,B 0,C 180,E1 -18755.493,E2 -18755.493} C_VEL
LIN {X 0,Y 249.348,Z 259.15,A -85,B 0,C 180,E1 -18755.941,E2 -18755.941} C_VEL
LIN {X 0,Y 250.031,Z 263.102,A -85,B 0,C 180,E1 -18760.278,E2 -18760.278} C_VEL
LIN {X 0,Y 250.839,Z 267.3,A -85,B 0,C 180,E1 -18764.463,E2 -18764.463} C_VEL
LIN {X 0,Y 251.534,Z 270.965,A -85,B 0,C 180,E1 -18767.889,E2 -18767.889} C_VEL
LIN {X 0,Y 252.128,Z 274.861,A -85,B 0,C 180,E1 -18771.306,E2 -18771.306} C_VEL
LIN {X 0,Y 251.885,Z 278.317,A -85,B 0,C 180,E1 -18774.131,E2 -18774.131} C_VEL
LIN {X 0,Y 250.512,Z 284.22,A -85,B 0,C 180,E1 -18778.734,E2 -18778.734} C_VEL
LIN {X 0,Y 250.108,Z 286.292,A -85,B 0,C 180,E1 -18780.269,E2 -18780.269} C_VEL
LIN {X 0,Y 253.338,Z 299.931,A -85,B 0,C 180,E1 -18781.415,E2 -18781.415} C_VEL
LIN {X 0,Y 255.387,Z 311.676,A -85,B 0,C 180,E1 -18782.608,E2 -18782.608} C_VEL
LIN {X 0,Y 256.658,Z 323.504,A -85,B 0,C 180,E1 -18784.016,E2 -18784.016} C_VEL
LIN {X 0,Y 257.067,Z 334.525,A -85,B 0,C 180,E1 -18785.551,E2 -18785.551} C_VEL
LIN {X 0,Y 256.898,Z 343.74,A -85,B 0,C 180,E1 -18787.056,E2 -18787.056} C_VEL
LIN {X 0,Y 254.554,Z 354.238,A -85,B 0,C 180,E1 -18788.966,E2 -18788.966} C_VEL
LIN {X 0,Y 252.466,Z 363.682,A -85,B 0,C 180,E1 -18791.169,E2 -18791.169} C_VEL
LIN {X 0,Y 250.871,Z 371.08,A -85,B 0,C 180,E1 -18793.313,E2 -18793.313} C_VEL
LIN {X 0,Y 249.375,Z 377.798,A -85,B 0,C 180,E1 -18795.724,E2 -18795.724} C_VEL
LIN {X 0,Y 248.11,Z 383.956,A -85,B 0,C 180,E1 -18798.564,E2 -18798.564} C_VEL
LIN {X 0,Y 247.497,Z 387.973,A -85,B 0,C 180,E1 -18801.015,E2 -18801.015} C_VEL
LIN {X 0,Y 247.172,Z 390.948,A -85,B 0,C 180,E1 -18803.47,E2 -18803.47} C_VEL
LIN {X 0,Y 247.081,Z 392.368,A -85,B 0,C 180,E1 -18805.105,E2 -18805.105} C_VEL
LIN {X 0,Y 247.092,Z 393.385,A -85,B 0,C 180,E1 -18806.739,E2 -18806.739} C_VEL
LIN {X 0,Y 247.106,Z 394.006,A -85,B 0,C 180,E1 -18808.37,E2 -18808.37} C_VEL
LIN {X 0,Y 247.178,Z 394.227,A -85,B 0,C 180,E1 -18810,E2 -18810} C_VEL
LIN {X 0,Y 247.106,Z 393.999,A -85,B 0,C 180,E1 -18811.63,E2 -18811.63} C_VEL
LIN {X 0,Y 247.09,Z 393.374,A -85,B 0,C 180,E1 -18813.261,E2 -18813.261} C_VEL
LIN {X 0,Y 247.088,Z 391.937,A -85,B 0,C 180,E1 -18815.427,E2 -18815.427} C_VEL
LIN {X 0,Y 247.345,Z 389.028,A -85,B 0,C 180,E1 -18818.168,E2 -18818.168} C_VEL
LIN {X 0,Y 247.847,Z 385.357,A -85,B 0,C 180,E1 -18820.622,E2 -18820.622} C_VEL
LIN {X 0,Y 248.69,Z 380.575,A -85,B 0,C 180,E1 -18823.067,E2 -18823.067} C_VEL
LIN {X 0,Y 250.371,Z 373.422,A -85,B 0,C 180,E1 -18825.884,E2 -18825.884} C_VEL
LIN {X 0,Y 252.154,Z 365.722,A -85,B 0,C 180,E1 -18828.257,E2 -18828.257} C_VEL
LIN {X 0,Y 253.755,Z 357.718,A -85,B 0,C 180,E1 -18830.255,E2 -18830.255} C_VEL
LIN {X 0,Y 255.925,Z 348.058,A -85,B 0,C 180,E1 -18832.185,E2 -18832.185} C_VEL
LIN {X 0,Y 257.015,Z 342.392,A -85,B 0,C 180,E1 -18833.147,E2 -18833.147} C_VEL
LIN {X 0,Y 256.973,Z 330.637,A -85,B 0,C 180,E1 -18834.998,E2 -18834.998} C_VEL
LIN {X 0,Y 256.264,Z 319.182,A -85,B 0,C 180,E1 -18836.497,E2 -18836.497} C_VEL
LIN {X 0,Y 254.728,Z 307.594,A -85,B 0,C 180,E1 -18837.796,E2 -18837.796} C_VEL
LIN {X 0,Y 252.132,Z 294.72,A -85,B 0,C 180,E1 -18839.026,E2 -18839.026} C_VEL
LIN {X 0,Y 250.109,Z 286.152,A -85,B 0,C 180,E1 -18839.715,E2 -18839.715} C_VEL
LIN {X 0,Y 251.32,Z 280.639,A -85,B 0,C 180,E1 -18844.007,E2 -18844.007} C_VEL
LIN {X 0,Y 252.087,Z 277.059,A -85,B 0,C 180,E1 -18846.827,E2 -18846.827} C_VEL
LIN {X 0,Y 251.981,Z 273.404,A -85,B 0,C 180,E1 -18849.904,E2 -18849.904} C_VEL
LIN {X 0,Y 251.051,Z 268.422,A -85,B 0,C 180,E1 -18854.416,E2 -18854.416} C_VEL
LIN {X 0,Y 250.123,Z 263.398,A -85,B 0,C 180,E1 -18859.346,E2 -18859.346} C_VEL
LIN {X 0,Y 249.403,Z 259.37,A -85,B 0,C 180,E1 -18863.718,E2 -18863.718} C_VEL
LIN {X 0,Y 249.03,Z 257.467,A -85,B 0,C 180,E1 -18866.126,E2 -18866.126} C_VEL
LIN {X 0,Y 249.005,Z 257.469,A -85,B 0,C 180,E1 -18869.467,E2 -18869.467} C_VEL
LIN {X 0,Y 249.028,Z 257.466,A -85,B 0,C 180,E1 -18873.157,E2 -18873.157} C_VEL
LIN {X 0,Y 249.013,Z 257.47,A -85,B 0,C 180,E1 -18876.726,E2 -18876.726} C_VEL
LIN {X 0,Y 249.103,Z 257.458,A -85,B 0,C 180,E1 -18880.211,E2 -18880.211} C_VEL
LIN {X 0,Y 249.246,Z 257.439,A -85,B 0,C 180,E1 -18883.622,E2 -18883.622} C_VEL
LIN {X 0,Y 249.246,Z 257.437,A -85,B 0,C 180,E1 -18888.616,E2 -18888.616} C_VEL
LIN {X 0,Y 249.448,Z 257.413,A -85,B 0,C 180,E1 -18891.902,E2 -18891.902} C_VEL
LIN {X 0,Y 249.297,Z 257.432,A -85,B 0,C 180,E1 -18895.149,E2 -18895.149} C_VEL
LIN {X 0,Y 249.679,Z 257.383,A -85,B 0,C 180,E1 -18898.387,E2 -18898.387} C_VEL
LIN {X 0,Y 249.663,Z 257.387,A -85,B 0,C 180,E1 -18901.613,E2 -18901.613} C_VEL
LIN {X 0,Y 249.434,Z 257.41,A -85,B 0,C 180,E1 -18906.703,E2 -18906.703} C_VEL
LIN {X 0,Y 249.346,Z 257.425,A -85,B 0,C 180,E1 -18909.736,E2 -18909.736} C_VEL
LIN {X 0,Y 249.179,Z 257.446,A -85,B 0,C 180,E1 -18914.705,E2 -18914.705} C_VEL
LIN {X 0,Y 249.112,Z 257.451,A -85,B 0,C 180,E1 -18918.08,E2 -18918.08} C_VEL
LIN {X 0,Y 249.084,Z 257.457,A -85,B 0,C 180,E1 -18921.519,E2 -18921.519} C_VEL
LIN {X 0,Y 249.088,Z 257.456,A -85,B 0,C 180,E1 -18925.46,E2 -18925.46} C_VEL
LIN {X 0,Y 249.04,Z 257.464,A -85,B 0,C 180,E1 -18928.974,E2 -18928.974} C_VEL
LIN {X 0,Y 249.03,Z 257.466,A -85,B 0,C 180,E1 -18932.426,E2 -18932.426} C_VEL
LIN {X 0,Y 249.052,Z 257.459,A -85,B 0,C 180,E1 -18936.342,E2 -18936.342} C_VEL
LIN {X 0,Y 249.009,Z 257.469,A -85,B 0,C 180,E1 -18940.478,E2 -18940.478} C_VEL
LIN {X 0,Y 249.005,Z 257.465,A -85,B 0,C 180,E1 -18944.879,E2 -18944.879} C_VEL
LIN {X 0,Y 249.019,Z 257.465,A -85,B 0,C 180,E1 -18947.363,E2 -18947.363} C_VEL
LIN {X 0,Y 248.982,Z 257.471,A -85,B 0,C 180,E1 -18951.611,E2 -18951.611} C_VEL
LIN {X 0,Y 248.882,Z 257.482,A -85,B 0,C 180,E1 -18953.629,E2 -18953.629} C_VEL
LIN {X 0,Y 248.856,Z 258.375,A -85,B 0,C 180,E1 -18955.609,E2 -18955.609} C_VEL
LIN {X 0,Y 248.726,Z 260.976,A -85,B 0,C 180,E1 -18959.428,E2 -18959.428} C_VEL
LIN {X 0,Y 248.733,Z 261.506,A -85,B 0,C 180,E1 -18960.192,E2 -18960.192} C_VEL
LIN {X 0,Y 251.04,Z 267.638,A -85,B 0,C 180,E1 -18960.847,E2 -18960.847} C_VEL
LIN {X 0,Y 254.821,Z 277.847,A -85,B 0,C 180,E1 -18962.039,E2 -18962.039} C_VEL
LIN {X 0,Y 258.1,Z 289.318,A -85,B 0,C 180,E1 -18963.52,E2 -18963.52} C_VEL
LIN {X 0,Y 260.185,Z 299.42,A -85,B 0,C 180,E1 -18964.977,E2 -18964.977} C_VEL
LIN {X 0,Y 260.759,Z 304.665,A -85,B 0,C 180,E1 -18965.782,E2 -18965.782} C_VEL
LIN {X 0,Y 258.751,Z 315.857,A -85,B 0,C 180,E1 -18967.441,E2 -18967.441} C_VEL
LIN {X 0,Y 256.951,Z 325.119,A -85,B 0,C 180,E1 -18969.171,E2 -18969.171} C_VEL
LIN {X 0,Y 254.992,Z 333.571,A -85,B 0,C 180,E1 -18971.104,E2 -18971.104} C_VEL
LIN {X 0,Y 252.978,Z 341.779,A -85,B 0,C 180,E1 -18973.455,E2 -18973.455} C_VEL
LIN {X 0,Y 251.644,Z 347.384,A -85,B 0,C 180,E1 -18975.442,E2 -18975.442} C_VEL
LIN {X 0,Y 250.117,Z 352.855,A -85,B 0,C 180,E1 -18977.834,E2 -18977.834} C_VEL
LIN {X 0,Y 249.067,Z 357.138,A -85,B 0,C 180,E1 -18980.252,E2 -18980.252} C_VEL
LIN {X 0,Y 248.547,Z 359.4,A -85,B 0,C 180,E1 -18981.872,E2 -18981.872} C_VEL
LIN {X 0,Y 248.147,Z 361.239,A -85,B 0,C 180,E1 -18983.495,E2 -18983.495} C_VEL
LIN {X 0,Y 247.765,Z 362.625,A -85,B 0,C 180,E1 -18985.118,E2 -18985.118} C_VEL
LIN {X 0,Y 247.356,Z 364.216,A -85,B 0,C 180,E1 -18988.372,E2 -18988.372} C_VEL
LIN {X 0,Y 247.324,Z 364.443,A -85,B 0,C 180,E1 -18990,E2 -18990} C_VEL
LIN {X 0,Y 247.5,Z 363.669,A -85,B 0,C 180,E1 -18993.255,E2 -18993.255} C_VEL
LIN {X 0,Y 248.124,Z 361.356,A -85,B 0,C 180,E1 -18996.505,E2 -18996.505} C_VEL
LIN {X 0,Y 248.742,Z 358.616,A -85,B 0,C 180,E1 -18998.858,E2 -18998.858} C_VEL
LIN {X 0,Y 249.676,Z 354.65,A -85,B 0,C 180,E1 -19001.364,E2 -19001.364} C_VEL
LIN {X 0,Y 251.001,Z 349.657,A -85,B 0,C 180,E1 -19003.768,E2 -19003.768} C_VEL
LIN {X 0,Y 252.619,Z 343.366,A -85,B 0,C 180,E1 -19006.153,E2 -19006.153} C_VEL
LIN {X 0,Y 254.571,Z 335.488,A -85,B 0,C 180,E1 -19008.511,E2 -19008.511} C_VEL
LIN {X 0,Y 256.946,Z 325.675,A -85,B 0,C 180,E1 -19010.829,E2 -19010.829} C_VEL
LIN {X 0,Y 258.812,Z 315.823,A -85,B 0,C 180,E1 -19012.685,E2 -19012.685} C_VEL
LIN {X 0,Y 260.887,Z 304.061,A -85,B 0,C 180,E1 -19014.422,E2 -19014.422} C_VEL
LIN {X 0,Y 259.274,Z 294.374,A -85,B 0,C 180,E1 -19015.896,E2 -19015.896} C_VEL
LIN {X 0,Y 256.364,Z 282.744,A -85,B 0,C 180,E1 -19017.478,E2 -19017.478} C_VEL
LIN {X 0,Y 252.24,Z 270.614,A -85,B 0,C 180,E1 -19018.942,E2 -19018.942} C_VEL
LIN {X 0,Y 248.861,Z 262.265,A -85,B 0,C 180,E1 -19019.858,E2 -19019.858} C_VEL
LIN {X 0,Y 248.727,Z 261.446,A -85,B 0,C 180,E1 -19019.981,E2 -19019.981} C_VEL
LIN {X 0,Y 248.808,Z 259.768,A -85,B 0,C 180,E1 -19022.458,E2 -19022.458} C_VEL
LIN {X 0,Y 248.885,Z 258.059,A -85,B 0,C 180,E1 -19025.025,E2 -19025.025} C_VEL
LIN {X 0,Y 248.881,Z 257.487,A -85,B 0,C 180,E1 -19026.371,E2 -19026.371} C_VEL
LIN {X 0,Y 248.99,Z 257.473,A -85,B 0,C 180,E1 -19030.35,E2 -19030.35} C_VEL
LIN {X 0,Y 249.01,Z 257.467,A -85,B 0,C 180,E1 -19032.792,E2 -19032.792} C_VEL
LIN {X 0,Y 249.018,Z 257.463,A -85,B 0,C 180,E1 -19037.363,E2 -19037.363} C_VEL
LIN {X 0,Y 249.046,Z 257.463,A -85,B 0,C 180,E1 -19042.2,E2 -19042.2} C_VEL
LIN {X 0,Y 249.045,Z 257.463,A -85,B 0,C 180,E1 -19045.639,E2 -19045.639} C_VEL
LIN {X 0,Y 249.003,Z 257.468,A -85,B 0,C 180,E1 -19049.466,E2 -19049.466} C_VEL
LIN {X 0,Y 249.036,Z 257.465,A -85,B 0,C 180,E1 -19053.158,E2 -19053.158} C_VEL
LIN {X 0,Y 249.056,Z 257.461,A -85,B 0,C 180,E1 -19056.73,E2 -19056.73} C_VEL
LIN {X 0,Y 249.085,Z 257.457,A -85,B 0,C 180,E1 -19060.209,E2 -19060.209} C_VEL
LIN {X 0,Y 249.197,Z 257.443,A -85,B 0,C 180,E1 -19063.619,E2 -19063.619} C_VEL
LIN {X 0,Y 249.253,Z 257.436,A -85,B 0,C 180,E1 -19068.616,E2 -19068.616} C_VEL
LIN {X 0,Y 249.486,Z 257.406,A -85,B 0,C 180,E1 -19071.903,E2 -19071.903} C_VEL
LIN {X 0,Y 249.287,Z 257.432,A -85,B 0,C 180,E1 -19075.148,E2 -19075.148} C_VEL
LIN {X 0,Y 249.662,Z 257.387,A -85,B 0,C 180,E1 -19078.387,E2 -19078.387} C_VEL
LIN {X 0,Y 249.677,Z 257.383,A -85,B 0,C 180,E1 -19081.613,E2 -19081.613} C_VEL
LIN {X 0,Y 249.449,Z 257.412,A -85,B 0,C 180,E1 -19086.471,E2 -19086.471} C_VEL
LIN {X 0,Y 249.345,Z 257.423,A -85,B 0,C 180,E1 -19089.736,E2 -19089.736} C_VEL
LIN {X 0,Y 249.207,Z 257.44,A -85,B 0,C 180,E1 -19094.703,E2 -19094.703} C_VEL
LIN {X 0,Y 249.139,Z 257.452,A -85,B 0,C 180,E1 -19098.077,E2 -19098.077} C_VEL
LIN {X 0,Y 249.08,Z 257.46,A -85,B 0,C 180,E1 -19101.519,E2 -19101.519} C_VEL
LIN {X 0,Y 249.05,Z 257.466,A -85,B 0,C 180,E1 -19105.442,E2 -19105.442} C_VEL
LIN {X 0,Y 249.037,Z 257.468,A -85,B 0,C 180,E1 -19108.974,E2 -19108.974} C_VEL
LIN {X 0,Y 249.042,Z 257.467,A -85,B 0,C 180,E1 -19113.387,E2 -19113.387} C_VEL
LIN {X 0,Y 249.117,Z 257.771,A -85,B 0,C 180,E1 -19114.349,E2 -19114.349} C_VEL
LIN {X 0,Y 249.348,Z 259.15,A -85,B 0,C 180,E1 -19115.941,E2 -19115.941} C_VEL
LIN {X 0,Y 248.896,Z 260.461,A -85,B 0,C 180,E1 -19117.258,E2 -19117.258} C_VEL
LIN {X 0,Y 246.461,Z 263.004,A -85,B 0,C 180,E1 -19119.398,E2 -19119.398} C_VEL
LIN {X 0,Y 244.38,Z 265.113,A -85,B 0,C 180,E1 -19121.135,E2 -19121.135} C_VEL
LIN {X 0,Y 243.576,Z 266.606,A -85,B 0,C 180,E1 -19122.478,E2 -19122.478} C_VEL
LIN {X 0,Y 243.562,Z 267.071,A -85,B 0,C 180,E1 -19122.933,E2 -19122.933} C_VEL
LIN {X 0,Y 244.409,Z 271.475,A -85,B 0,C 180,E1 -19127.233,E2 -19127.233} C_VEL
LIN {X 0,Y 245.063,Z 275.453,A -85,B 0,C 180,E1 -19130.882,E2 -19130.882} C_VEL
LIN {X 0,Y 244.997,Z 278.436,A -85,B 0,C 180,E1 -19133.438,E2 -19133.438} C_VEL
LIN {X 0,Y 243.715,Z 283.777,A -85,B 0,C 180,E1 -19137.759,E2 -19137.759} C_VEL
LIN {X 0,Y 243.28,Z 285.731,A -85,B 0,C 180,E1 -19139.325,E2 -19139.325} C_VEL
LIN {X 0,Y 245.517,Z 294.86,A -85,B 0,C 180,E1 -19140.116,E2 -19140.116} C_VEL
LIN {X 0,Y 248.115,Z 307.74,A -85,B 0,C 180,E1 -19141.413,E2 -19141.413} C_VEL
LIN {X 0,Y 249.668,Z 319.414,A -85,B 0,C 180,E1 -19142.789,E2 -19142.789} C_VEL
LIN {X 0,Y 250.33,Z 330.345,A -85,B 0,C 180,E1 -19144.282,E2 -19144.282} C_VEL
LIN {X 0,Y 250.306,Z 340.918,A -85,B 0,C 180,E1 -19145.976,E2 -19145.976} C_VEL
LIN {X 0,Y 249.881,Z 345.63,A -85,B 0,C 180,E1 -19146.812,E2 -19146.812} C_VEL
LIN {X 0,Y 247.488,Z 355.615,A -85,B 0,C 180,E1 -19148.773,E2 -19148.773} C_VEL
LIN {X 0,Y 245.517,Z 364.049,A -85,B 0,C 180,E1 -19150.846,E2 -19150.846} C_VEL
LIN {X 0,Y 244.055,Z 370.653,A -85,B 0,C 180,E1 -19152.833,E2 -19152.833} C_VEL
LIN {X 0,Y 242.469,Z 377.37,A -85,B 0,C 180,E1 -19155.308,E2 -19155.308} C_VEL
LIN {X 0,Y 241.123,Z 383.527,A -85,B 0,C 180,E1 -19158.228,E2 -19158.228} C_VEL
LIN {X 0,Y 240.441,Z 387.543,A -85,B 0,C 180,E1 -19160.749,E2 -19160.749} C_VEL
LIN {X 0,Y 240.087,Z 390.519,A -85,B 0,C 180,E1 -19163.276,E2 -19163.276} C_VEL
LIN {X 0,Y 240.009,Z 391.941,A -85,B 0,C 180,E1 -19164.96,E2 -19164.96} C_VEL
LIN {X 0,Y 240.006,Z 392.958,A -85,B 0,C 180,E1 -19166.643,E2 -19166.643} C_VEL
LIN {X 0,Y 240.033,Z 393.58,A -85,B 0,C 180,E1 -19168.322,E2 -19168.322} C_VEL
LIN {X 0,Y 240.1,Z 393.801,A -85,B 0,C 180,E1 -19170,E2 -19170} C_VEL
LIN {X 0,Y 240.033,Z 393.572,A -85,B 0,C 180,E1 -19171.678,E2 -19171.678} C_VEL
LIN {X 0,Y 240.003,Z 392.947,A -85,B 0,C 180,E1 -19173.358,E2 -19173.358} C_VEL
LIN {X 0,Y 239.989,Z 391.725,A -85,B 0,C 180,E1 -19175.326,E2 -19175.326} C_VEL
LIN {X 0,Y 240.297,Z 388.598,A -85,B 0,C 180,E1 -19178.409,E2 -19178.409} C_VEL
LIN {X 0,Y 240.843,Z 384.927,A -85,B 0,C 180,E1 -19180.934,E2 -19180.934} C_VEL
LIN {X 0,Y 241.738,Z 380.143,A -85,B 0,C 180,E1 -19183.449,E2 -19183.449} C_VEL
LIN {X 0,Y 243.258,Z 374.12,A -85,B 0,C 180,E1 -19185.931,E2 -19185.931} C_VEL
LIN {X 0,Y 245.06,Z 366.623,A -85,B 0,C 180,E1 -19188.389,E2 -19188.389} C_VEL
LIN {X 0,Y 246.689,Z 358.98,A -85,B 0,C 180,E1 -19190.426,E2 -19190.426} C_VEL
LIN {X 0,Y 248.885,Z 349.757,A -85,B 0,C 180,E1 -19192.409,E2 -19192.409} C_VEL
LIN {X 0,Y 250.227,Z 343.139,A -85,B 0,C 180,E1 -19193.593,E2 -19193.593} C_VEL
LIN {X 0,Y 250.291,Z 331.433,A -85,B 0,C 180,E1 -19195.531,E2 -19195.531} C_VEL
LIN {X 0,Y 249.767,Z 321.079,A -85,B 0,C 180,E1 -19196.973,E2 -19196.973} C_VEL
LIN {X 0,Y 248.456,Z 310.033,A -85,B 0,C 180,E1 -19198.307,E2 -19198.307} C_VEL
LIN {X 0,Y 246.016,Z 297.078,A -85,B 0,C 180,E1 -19199.641,E2 -19199.641} C_VEL
LIN {X 0,Y 243.272,Z 285.643,A -85,B 0,C 180,E1 -19200.678,E2 -19200.678} C_VEL
LIN {X 0,Y 244.593,Z 280.205,A -85,B 0,C 180,E1 -19205.077,E2 -19205.077} C_VEL
LIN {X 0,Y 245.07,Z 277.825,A -85,B 0,C 180,E1 -19207.03,E2 -19207.03} C_VEL
LIN {X 0,Y 244.905,Z 274.176,A -85,B 0,C 180,E1 -19210.216,E2 -19210.216} C_VEL
LIN {X 0,Y 244.155,Z 270.121,A -85,B 0,C 180,E1 -19213.976,E2 -19213.976} C_VEL
LIN {X 0,Y 243.265,Z 265.466,A -85,B 0,C 180,E1 -19218.691,E2 -19218.691} C_VEL
LIN {X 0,Y 242.627,Z 261.919,A -85,B 0,C 180,E1 -19222.534,E2 -19222.534} C_VEL
LIN {X 0,Y 242.034,Z 258.583,A -85,B 0,C 180,E1 -19226.516,E2 -19226.516} C_VEL
LIN {X 0,Y 241.994,Z 258.34,A -85,B 0,C 180,E1 -19227.376,E2 -19227.376} C_VEL
LIN {X 0,Y 241.979,Z 258.345,A -85,B 0,C 180,E1 -19230.613,E2 -19230.613} C_VEL
LIN {X 0,Y 241.999,Z 258.343,A -85,B 0,C 180,E1 -19234.197,E2 -19234.197} C_VEL
LIN {X 0,Y 242.019,Z 258.341,A -85,B 0,C 180,E1 -19238.319,E2 -19238.319} C_VEL
LIN {X 0,Y 242.167,Z 258.32,A -85,B 0,C 180,E1 -19243.278,E2 -19243.278} C_VEL
LIN {X 0,Y 242.183,Z 258.318,A -85,B 0,C 180,E1 -19248.28,E2 -19248.28} C_VEL
LIN {X 0,Y 242.396,Z 258.294,A -85,B 0,C 180,E1 -19251.665,E2 -19251.665} C_VEL
LIN {X 0,Y 242.258,Z 258.308,A -85,B 0,C 180,E1 -19255.007,E2 -19255.007} C_VEL
LIN {X 0,Y 242.639,Z 258.26,A -85,B 0,C 180,E1 -19258.34,E2 -19258.34} C_VEL
LIN {X 0,Y 242.624,Z 258.264,A -85,B 0,C 180,E1 -19261.66,E2 -19261.66} C_VEL
LIN {X 0,Y 242.416,Z 258.286,A -85,B 0,C 180,E1 -19266.675,E2 -19266.675} C_VEL
LIN {X 0,Y 242.269,Z 258.306,A -85,B 0,C 180,E1 -19270.024,E2 -19270.024} C_VEL
LIN {X 0,Y 242.138,Z 258.323,A -85,B 0,C 180,E1 -19275.143,E2 -19275.143} C_VEL
LIN {X 0,Y 242.05,Z 258.333,A -85,B 0,C 180,E1 -19278.626,E2 -19278.626} C_VEL
LIN {X 0,Y 242.006,Z 258.339,A -85,B 0,C 180,E1 -19282.181,E2 -19282.181} C_VEL
LIN {X 0,Y 242.035,Z 258.334,A -85,B 0,C 180,E1 -19285.821,E2 -19285.821} C_VEL
LIN {X 0,Y 241.972,Z 258.343,A -85,B 0,C 180,E1 -19289.588,E2 -19289.588} C_VEL
LIN {X 0,Y 241.983,Z 258.341,A -85,B 0,C 180,E1 -19293.493,E2 -19293.493} C_VEL
LIN {X 0,Y 241.993,Z 258.34,A -85,B 0,C 180,E1 -19297.581,E2 -19297.581} C_VEL
LIN {X 0,Y 241.941,Z 258.348,A -85,B 0,C 180,E1 -19301.922,E2 -19301.922} C_VEL
LIN {X 0,Y 241.937,Z 258.347,A -85,B 0,C 180,E1 -19306.571,E2 -19306.571} C_VEL
LIN {X 0,Y 241.935,Z 258.349,A -85,B 0,C 180,E1 -19310.276,E2 -19310.276} C_VEL
LIN {X 0,Y 241.908,Z 258.351,A -85,B 0,C 180,E1 -19312.403,E2 -19312.403} C_VEL
LIN {X 0,Y 241.863,Z 258.831,A -85,B 0,C 180,E1 -19314.468,E2 -19314.468} C_VEL
LIN {X 0,Y 241.768,Z 261.411,A -85,B 0,C 180,E1 -19318.449,E2 -19318.449} C_VEL
LIN {X 0,Y 241.731,Z 262.038,A -85,B 0,C 180,E1 -19319.27,E2 -19319.27} C_VEL
LIN {X 0,Y 242.824,Z 265.088,A -85,B 0,C 180,E1 -19319.586,E2 -19319.586} C_VEL
LIN {X 0,Y 247.371,Z 276.449,A -85,B 0,C 180,E1 -19320.968,E2 -19320.968} C_VEL
LIN {X 0,Y 250.825,Z 287.898,A -85,B 0,C 180,E1 -19322.477,E2 -19322.477} C_VEL
LIN {X 0,Y 253.264,Z 298.844,A -85,B 0,C 180,E1 -19324.096,E2 -19324.096} C_VEL
LIN {X 0,Y 254.237,Z 305.293,A -85,B 0,C 180,E1 -19325.149,E2 -19325.149} C_VEL
LIN {X 0,Y 252.173,Z 316.63,A -85,B 0,C 180,E1 -19326.883,E2 -19326.883} C_VEL
LIN {X 0,Y 250.35,Z 325.548,A -85,B 0,C 180,E1 -19328.595,E2 -19328.595} C_VEL
LIN {X 0,Y 248.312,Z 333.999,A -85,B 0,C 180,E1 -19330.575,E2 -19330.575} C_VEL
LIN {X 0,Y 246.209,Z 342.207,A -85,B 0,C 180,E1 -19332.987,E2 -19332.987} C_VEL
LIN {X 0,Y 244.795,Z 347.812,A -85,B 0,C 180,E1 -19335.025,E2 -19335.025} C_VEL
LIN {X 0,Y 243.198,Z 353.283,A -85,B 0,C 180,E1 -19337.482,E2 -19337.482} C_VEL
LIN {X 0,Y 242.074,Z 357.566,A -85,B 0,C 180,E1 -19339.968,E2 -19339.968} C_VEL
LIN {X 0,Y 241.523,Z 359.829,A -85,B 0,C 180,E1 -19341.634,E2 -19341.634} C_VEL
LIN {X 0,Y 241.103,Z 361.667,A -85,B 0,C 180,E1 -19343.304,E2 -19343.304} C_VEL
LIN {X 0,Y 240.721,Z 363.051,A -85,B 0,C 180,E1 -19344.975,E2 -19344.975} C_VEL
LIN {X 0,Y 240.279,Z 364.643,A -85,B 0,C 180,E1 -19348.324,E2 -19348.324} C_VEL
LIN {X 0,Y 240.242,Z 364.87,A -85,B 0,C 180,E1 -19350,E2 -19350} C_VEL
LIN {X 0,Y 240.435,Z 364.095,A -85,B 0,C 180,E1 -19353.351,E2 -19353.351} C_VEL
LIN {X 0,Y 241.08,Z 361.783,A -85,B 0,C 180,E1 -19356.696,E2 -19356.696} C_VEL
LIN {X 0,Y 241.786,Z 358.936,A -85,B 0,C 180,E1 -19359.199,E2 -19359.199} C_VEL
LIN {X 0,Y 242.737,Z 355.075,A -85,B 0,C 180,E1 -19361.693,E2 -19361.693} C_VEL
LIN {X 0,Y 244.131,Z 350.082,A -85,B 0,C 180,E1 -19364.164,E2 -19364.164} C_VEL
LIN {X 0,Y 245.818,Z 343.79,A -85,B 0,C 180,E1 -19366.613,E2 -19366.613} C_VEL
LIN {X 0,Y 247.873,Z 335.911,A -85,B 0,C 180,E1 -19369.03,E2 -19369.03} C_VEL
LIN {X 0,Y 250.352,Z 326.098,A -85,B 0,C 180,E1 -19371.404,E2 -19371.404} C_VEL
LIN {X 0,Y 252.372,Z 315.803,A -85,B 0,C 180,E1 -19373.38,E2 -19373.38} C_VEL
LIN {X 0,Y 254.259,Z 305.981,A -85,B 0,C 180,E1 -19374.87,E2 -19374.87} C_VEL
LIN {X 0,Y 253.212,Z 298.261,A -85,B 0,C 180,E1 -19376.119,E2 -19376.119} C_VEL
LIN {X 0,Y 250.605,Z 286.949,A -85,B 0,C 180,E1 -19377.78,E2 -19377.78} C_VEL
LIN {X 0,Y 246.934,Z 275.361,A -85,B 0,C 180,E1 -19379.309,E2 -19379.309} C_VEL
LIN {X 0,Y 242.628,Z 264.7,A -85,B 0,C 180,E1 -19380.599,E2 -19380.599} C_VEL
LIN {X 0,Y 241.73,Z 261.937,A -85,B 0,C 180,E1 -19380.9,E2 -19380.9} C_VEL
LIN {X 0,Y 241.81,Z 260.225,A -85,B 0,C 180,E1 -19383.519,E2 -19383.519} C_VEL
LIN {X 0,Y 241.853,Z 258.924,A -85,B 0,C 180,E1 -19385.545,E2 -19385.545} C_VEL
LIN {X 0,Y 241.951,Z 258.351,A -85,B 0,C 180,E1 -19388.346,E2 -19388.346} C_VEL
LIN {X 0,Y 241.934,Z 258.349,A -85,B 0,C 180,E1 -19391.923,E2 -19391.923} C_VEL
LIN {X 0,Y 241.936,Z 258.344,A -85,B 0,C 180,E1 -19396.571,E2 -19396.571} C_VEL
LIN {X 0,Y 241.958,Z 258.346,A -85,B 0,C 180,E1 -19400.281,E2 -19400.281} C_VEL
LIN {X 0,Y 241.99,Z 258.341,A -85,B 0,C 180,E1 -19404.489,E2 -19404.489} C_VEL
LIN {X 0,Y 241.954,Z 258.343,A -85,B 0,C 180,E1 -19408.477,E2 -19408.477} C_VEL
LIN {X 0,Y 241.969,Z 258.343,A -85,B 0,C 180,E1 -19412.308,E2 -19412.308} C_VEL
LIN {X 0,Y 242.026,Z 258.337,A -85,B 0,C 180,E1 -19416.013,E2 -19416.013} C_VEL
LIN {X 0,Y 242.021,Z 258.338,A -85,B 0,C 180,E1 -19419.606,E2 -19419.606} C_VEL
LIN {X 0,Y 242.117,Z 258.327,A -85,B 0,C 180,E1 -19423.316,E2 -19423.316} C_VEL
LIN {X 0,Y 242.186,Z 258.316,A -85,B 0,C 180,E1 -19428.28,E2 -19428.28} C_VEL
LIN {X 0,Y 242.437,Z 258.284,A -85,B 0,C 180,E1 -19431.666,E2 -19431.666} C_VEL
LIN {X 0,Y 242.249,Z 258.309,A -85,B 0,C 180,E1 -19435.007,E2 -19435.007} C_VEL
LIN {X 0,Y 242.622,Z 258.264,A -85,B 0,C 180,E1 -19438.34,E2 -19438.34} C_VEL
LIN {X 0,Y 242.637,Z 258.26,A -85,B 0,C 180,E1 -19441.66,E2 -19441.66} C_VEL
LIN {X 0,Y 242.419,Z 258.287,A -85,B 0,C 180,E1 -19446.659,E2 -19446.659} C_VEL
LIN {X 0,Y 242.269,Z 258.305,A -85,B 0,C 180,E1 -19450.024,E2 -19450.024} C_VEL
LIN {X 0,Y 242.169,Z 258.316,A -85,B 0,C 180,E1 -19455.141,E2 -19455.141} C_VEL
LIN {X 0,Y 242.07,Z 258.332,A -85,B 0,C 180,E1 -19458.624,E2 -19458.624} C_VEL
LIN {X 0,Y 241.99,Z 258.344,A -85,B 0,C 180,E1 -19462.182,E2 -19462.182} C_VEL
LIN {X 0,Y 241.988,Z 258.346,A -85,B 0,C 180,E1 -19465.826,E2 -19465.826} C_VEL
LIN {X 0,Y 241.969,Z 258.351,A -85,B 0,C 180,E1 -19469.588,E2 -19469.588} C_VEL
LIN {X 0,Y 242.011,Z 258.44,A -85,B 0,C 180,E1 -19473.232,E2 -19473.232} C_VEL
LIN {X 0,Y 242.42,Z 260.622,A -85,B 0,C 180,E1 -19475.897,E2 -19475.897} C_VEL
LIN {X 0,Y 242.955,Z 263.867,A -85,B 0,C 180,E1 -19479.524,E2 -19479.524} C_VEL
LIN {X 0,Y 243.562,Z 267.071,A -85,B 0,C 180,E1 -19482.933,E2 -19482.933} C_VEL
LIN {X 0,Y 243.129,Z 268.544,A -85,B 0,C 180,E1 -19484.276,E2 -19484.276} C_VEL
LIN {X 0,Y 240.745,Z 271.283,A -85,B 0,C 180,E1 -19486.461,E2 -19486.461} C_VEL
LIN {X 0,Y 238.714,Z 273.524,A -85,B 0,C 180,E1 -19488.236,E2 -19488.236} C_VEL
LIN {X 0,Y 237.942,Z 275.132,A -85,B 0,C 180,E1 -19489.607,E2 -19489.607} C_VEL
LIN {X 0,Y 237.937,Z 275.641,A -85,B 0,C 180,E1 -19490.071,E2 -19490.071} C_VEL
LIN {X 0,Y 238.033,Z 278.747,A -85,B 0,C 180,E1 -19492.862,E2 -19492.862} C_VEL
LIN {X 0,Y 237.137,Z 282.555,A -85,B 0,C 180,E1 -19496.082,E2 -19496.082} C_VEL
LIN {X 0,Y 236.454,Z 285.287,A -85,B 0,C 180,E1 -19498.348,E2 -19498.348} C_VEL
LIN {X 0,Y 238.681,Z 294.125,A -85,B 0,C 180,E1 -19499.15,E2 -19499.15} C_VEL
LIN {X 0,Y 241.26,Z 306.47,A -85,B 0,C 180,E1 -19500.449,E2 -19500.449} C_VEL
LIN {X 0,Y 242.879,Z 318.279,A -85,B 0,C 180,E1 -19501.884,E2 -19501.884} C_VEL
LIN {X 0,Y 243.601,Z 329.274,A -85,B 0,C 180,E1 -19503.427,E2 -19503.427} C_VEL
LIN {X 0,Y 243.603,Z 340.478,A -85,B 0,C 180,E1 -19505.271,E2 -19505.271} C_VEL
LIN {X 0,Y 243.324,Z 345.203,A -85,B 0,C 180,E1 -19506.149,E2 -19506.149} C_VEL
LIN {X 0,Y 240.848,Z 355.188,A -85,B 0,C 180,E1 -19508.158,E2 -19508.158} C_VEL
LIN {X 0,Y 238.597,Z 364.365,A -85,B 0,C 180,E1 -19510.489,E2 -19510.489} C_VEL
LIN {X 0,Y 236.914,Z 371.468,A -85,B 0,C 180,E1 -19512.744,E2 -19512.744} C_VEL
LIN {X 0,Y 235.324,Z 377.945,A -85,B 0,C 180,E1 -19515.294,E2 -19515.294} C_VEL
LIN {X 0,Y 234.131,Z 383.098,A -85,B 0,C 180,E1 -19517.871,E2 -19517.871} C_VEL
LIN {X 0,Y 233.409,Z 387.115,A -85,B 0,C 180,E1 -19520.468,E2 -19520.468} C_VEL
LIN {X 0,Y 233.011,Z 390.091,A -85,B 0,C 180,E1 -19523.071,E2 -19523.071} C_VEL
LIN {X 0,Y 232.923,Z 391.513,A -85,B 0,C 180,E1 -19524.807,E2 -19524.807} C_VEL
LIN {X 0,Y 232.923,Z 392.531,A -85,B 0,C 180,E1 -19526.541,E2 -19526.541} C_VEL
LIN {X 0,Y 232.961,Z 393.154,A -85,B 0,C 180,E1 -19528.271,E2 -19528.271} C_VEL
LIN {X 0,Y 233.024,Z 393.375,A -85,B 0,C 180,E1 -19530,E2 -19530} C_VEL
LIN {X 0,Y 232.961,Z 393.146,A -85,B 0,C 180,E1 -19531.729,E2 -19531.729} C_VEL
LIN {X 0,Y 232.919,Z 392.519,A -85,B 0,C 180,E1 -19533.46,E2 -19533.46} C_VEL
LIN {X 0,Y 232.913,Z 391.437,A -85,B 0,C 180,E1 -19535.282,E2 -19535.282} C_VEL
LIN {X 0,Y 233.009,Z 390.066,A -85,B 0,C 180,E1 -19536.93,E2 -19536.93} C_VEL
LIN {X 0,Y 233.404,Z 387.078,A -85,B 0,C 180,E1 -19539.533,E2 -19539.533} C_VEL
LIN {X 0,Y 234.132,Z 383.046,A -85,B 0,C 180,E1 -19542.13,E2 -19542.13} C_VEL
LIN {X 0,Y 235.554,Z 376.868,A -85,B 0,C 180,E1 -19545.134,E2 -19545.134} C_VEL
LIN {X 0,Y 237.268,Z 370.138,A -85,B 0,C 180,E1 -19547.675,E2 -19547.675} C_VEL
LIN {X 0,Y 239.252,Z 361.877,A -85,B 0,C 180,E1 -19550.166,E2 -19550.166} C_VEL
LIN {X 0,Y 241.308,Z 353.247,A -85,B 0,C 180,E1 -19552.249,E2 -19552.249} C_VEL
LIN {X 0,Y 243.458,Z 343.886,A -85,B 0,C 180,E1 -19554.064,E2 -19554.064} C_VEL
LIN {X 0,Y 243.616,Z 332.193,A -85,B 0,C 180,E1 -19556.091,E2 -19556.091} C_VEL
LIN {X 0,Y 243.106,Z 320.844,A -85,B 0,C 180,E1 -19557.745,E2 -19557.745} C_VEL
LIN {X 0,Y 241.634,Z 308.916,A -85,B 0,C 180,E1 -19559.242,E2 -19559.242} C_VEL
LIN {X 0,Y 239.254,Z 296.627,A -85,B 0,C 180,E1 -19560.565,E2 -19560.565} C_VEL
LIN {X 0,Y 236.471,Z 285.21,A -85,B 0,C 180,E1 -19561.65,E2 -19561.65} C_VEL
LIN {X 0,Y 237.821,Z 279.755,A -85,B 0,C 180,E1 -19566.231,E2 -19566.231} C_VEL
LIN {X 0,Y 238.081,Z 277.367,A -85,B 0,C 180,E1 -19568.31,E2 -19568.31} C_VEL
LIN {X 0,Y 237.843,Z 274.91,A -85,B 0,C 180,E1 -19570.548,E2 -19570.548} C_VEL
LIN {X 0,Y 237.013,Z 270.719,A -85,B 0,C 180,E1 -19574.63,E2 -19574.63} C_VEL
LIN {X 0,Y 236.208,Z 266.448,A -85,B 0,C 180,E1 -19579.112,E2 -19579.112} C_VEL
LIN {X 0,Y 235.541,Z 262.425,A -85,B 0,C 180,E1 -19583.671,E2 -19583.671} C_VEL
LIN {X 0,Y 234.935,Z 259.217,A -85,B 0,C 180,E1 -19587.928,E2 -19587.928} C_VEL
LIN {X 0,Y 234.902,Z 259.224,A -85,B 0,C 180,E1 -19591.399,E2 -19591.399} C_VEL
LIN {X 0,Y 234.918,Z 259.225,A -85,B 0,C 180,E1 -19595.239,E2 -19595.239} C_VEL
LIN {X 0,Y 234.993,Z 259.215,A -85,B 0,C 180,E1 -19598.968,E2 -19598.968} C_VEL
LIN {X 0,Y 235.099,Z 259.2,A -85,B 0,C 180,E1 -19603.06,E2 -19603.06} C_VEL
LIN {X 0,Y 235.117,Z 259.198,A -85,B 0,C 180,E1 -19607.922,E2 -19607.922} C_VEL
LIN {X 0,Y 235.328,Z 259.172,A -85,B 0,C 180,E1 -19611.412,E2 -19611.412} C_VEL
LIN {X 0,Y 235.37,Z 259.165,A -85,B 0,C 180,E1 -19613.14,E2 -19613.14} C_VEL
LIN {X 0,Y 235.599,Z 259.137,A -85,B 0,C 180,E1 -19618.291,E2 -19618.291} C_VEL
LIN {X 0,Y 235.583,Z 259.141,A -85,B 0,C 180,E1 -19621.71,E2 -19621.71} C_VEL
LIN {X 0,Y 235.368,Z 259.165,A -85,B 0,C 180,E1 -19626.86,E2 -19626.86} C_VEL
LIN {X 0,Y 235.215,Z 259.185,A -85,B 0,C 180,E1 -19630.328,E2 -19630.328} C_VEL
LIN {X 0,Y 235.083,Z 259.202,A -85,B 0,C 180,E1 -19635.609,E2 -19635.609} C_VEL
LIN {X 0,Y 234.991,Z 259.214,A -85,B 0,C 180,E1 -19639.207,E2 -19639.207} C_VEL
LIN {X 0,Y 234.949,Z 259.218,A -85,B 0,C 180,E1 -19642.884,E2 -19642.884} C_VEL
LIN {X 0,Y 234.948,Z 259.219,A -85,B 0,C 180,E1 -19646.66,E2 -19646.66} C_VEL
LIN {X 0,Y 234.902,Z 259.225,A -85,B 0,C 180,E1 -19650.572,E2 -19650.572} C_VEL
LIN {X 0,Y 234.934,Z 259.22,A -85,B 0,C 180,E1 -19654.638,E2 -19654.638} C_VEL
LIN {X 0,Y 234.945,Z 259.216,A -85,B 0,C 180,E1 -19658.944,E2 -19658.944} C_VEL
LIN {X 0,Y 234.89,Z 259.226,A -85,B 0,C 180,E1 -19663.486,E2 -19663.486} C_VEL
LIN {X 0,Y 234.89,Z 259.225,A -85,B 0,C 180,E1 -19666.514,E2 -19666.514} C_VEL
LIN {X 0,Y 234.889,Z 259.225,A -85,B 0,C 180,E1 -19671.072,E2 -19671.072} C_VEL
LIN {X 0,Y 234.79,Z 259.302,A -85,B 0,C 180,E1 -19673.225,E2 -19673.225} C_VEL
LIN {X 0,Y 234.798,Z 261.876,A -85,B 0,C 180,E1 -19677.399,E2 -19677.399} C_VEL
LIN {X 0,Y 234.771,Z 262.415,A -85,B 0,C 180,E1 -19678.236,E2 -19678.236} C_VEL
LIN {X 0,Y 235.951,Z 265.662,A -85,B 0,C 180,E1 -19678.605,E2 -19678.605} C_VEL
LIN {X 0,Y 240.504,Z 276.97,A -85,B 0,C 180,E1 -19680.059,E2 -19680.059} C_VEL
LIN {X 0,Y 244.023,Z 288.233,A -85,B 0,C 180,E1 -19681.628,E2 -19681.628} C_VEL
LIN {X 0,Y 246.548,Z 299.301,A -85,B 0,C 180,E1 -19683.335,E2 -19683.335} C_VEL
LIN {X 0,Y 247.623,Z 306.969,A -85,B 0,C 180,E1 -19684.636,E2 -19684.636} C_VEL
LIN {X 0,Y 245.516,Z 317.857,A -85,B 0,C 180,E1 -19686.374,E2 -19686.374} C_VEL
LIN {X 0,Y 243.36,Z 327.774,A -85,B 0,C 180,E1 -19688.394,E2 -19688.394} C_VEL
LIN {X 0,Y 241.257,Z 335.901,A -85,B 0,C 180,E1 -19690.427,E2 -19690.427} C_VEL
LIN {X 0,Y 239.115,Z 343.854,A -85,B 0,C 180,E1 -19692.907,E2 -19692.907} C_VEL
LIN {X 0,Y 237.336,Z 350.231,A -85,B 0,C 180,E1 -19695.421,E2 -19695.421} C_VEL
LIN {X 0,Y 235.845,Z 355.288,A -85,B 0,C 180,E1 -19697.96,E2 -19697.96} C_VEL
LIN {X 0,Y 234.797,Z 359.205,A -85,B 0,C 180,E1 -19700.524,E2 -19700.524} C_VEL
LIN {X 0,Y 234.063,Z 362.094,A -85,B 0,C 180,E1 -19703.102,E2 -19703.102} C_VEL
LIN {X 0,Y 233.68,Z 363.478,A -85,B 0,C 180,E1 -19704.823,E2 -19704.823} C_VEL
LIN {X 0,Y 233.203,Z 365.069,A -85,B 0,C 180,E1 -19708.273,E2 -19708.273} C_VEL
LIN {X 0,Y 233.162,Z 365.296,A -85,B 0,C 180,E1 -19710,E2 -19710} C_VEL
LIN {X 0,Y 233.372,Z 364.521,A -85,B 0,C 180,E1 -19713.453,E2 -19713.453} C_VEL
LIN {X 0,Y 233.666,Z 363.557,A -85,B 0,C 180,E1 -19715.177,E2 -19715.177} C_VEL
LIN {X 0,Y 234.38,Z 360.792,A -85,B 0,C 180,E1 -19718.299,E2 -19718.299} C_VEL
LIN {X 0,Y 235.42,Z 356.904,A -85,B 0,C 180,E1 -19721.189,E2 -19721.189} C_VEL
LIN {X 0,Y 236.723,Z 352.297,A -85,B 0,C 180,E1 -19723.739,E2 -19723.739} C_VEL
LIN {X 0,Y 238.687,Z 345.345,A -85,B 0,C 180,E1 -19726.683,E2 -19726.683} C_VEL
LIN {X 0,Y 240.8,Z 337.8,A -85,B 0,C 180,E1 -19729.168,E2 -19729.168} C_VEL
LIN {X 0,Y 243.301,Z 328.292,A -85,B 0,C 180,E1 -19731.611,E2 -19731.611} C_VEL
LIN {X 0,Y 245.435,Z 318.487,A -85,B 0,C 180,E1 -19733.634,E2 -19733.634} C_VEL
LIN {X 0,Y 247.558,Z 307.72,A -85,B 0,C 180,E1 -19735.383,E2 -19735.383} C_VEL
LIN {X 0,Y 247.551,Z 305.493,A -85,B 0,C 180,E1 -19735.742,E2 -19735.742} C_VEL
LIN {X 0,Y 245.654,Z 294.782,A -85,B 0,C 180,E1 -19737.514,E2 -19737.514} C_VEL
LIN {X 0,Y 242.736,Z 283.608,A -85,B 0,C 180,E1 -19739.169,E2 -19739.169} C_VEL
